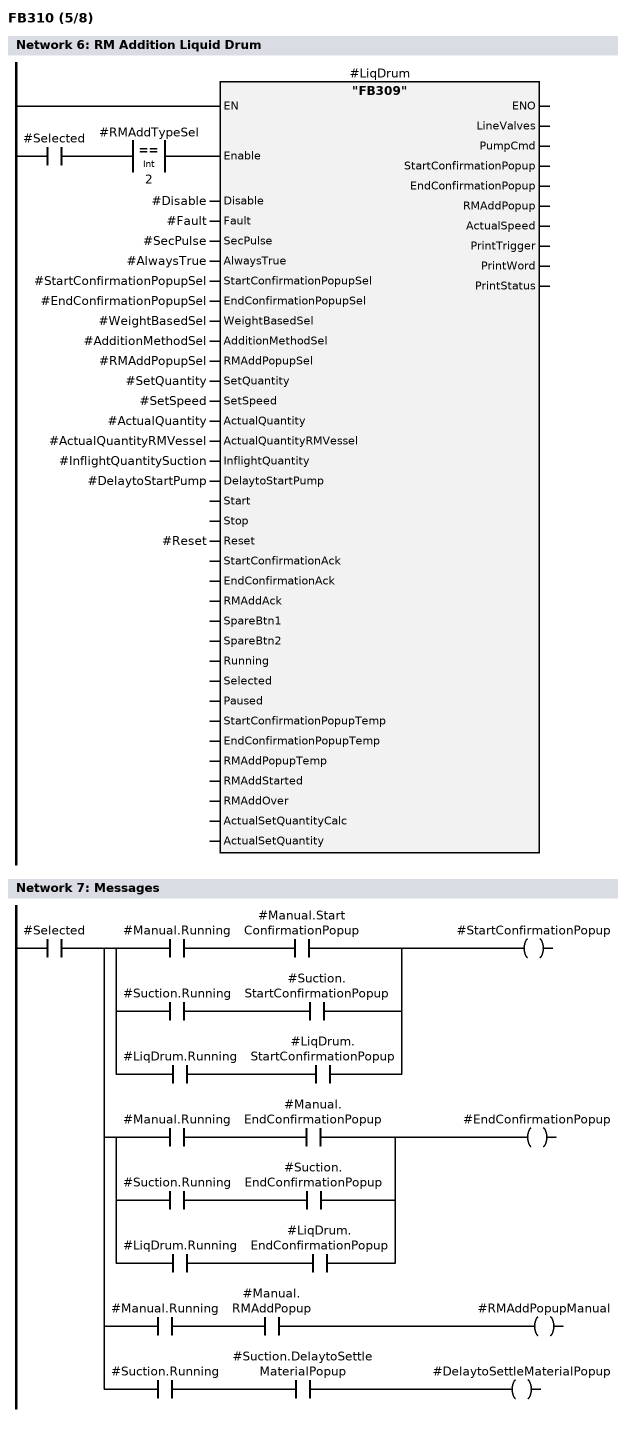
   RUNG wire#powerrail
      #LiqDrum(Enable := wire#w1, Disable := #Disable, Fault := #Fault, SecPulse := #SecPulse, AlwaysTrue := #AlwaysTrue, StartConfirmationPopupSel := #StartConfirmationPopupSel, EndConfirmationPopupSel := #EndConfirmationPopupSel, WeightBasedSel := #WeightBasedSel, AdditionMethodSel := #AdditionMethodSel, RMAddPopupSel := #RMAddPopupSel, SetQuantity := #SetQuantity, SetSpeed := #SetSpeed, ActualQuantity := #ActualQuantity, ActualQuantityRMVessel := #ActualQuantityRMVessel, InflightQuantity := #InflightQuantitySuction, DelaytoStartPump := #DelaytoStartPump, Start :=, Stop :=, Reset := #Reset, StartConfirmationAck :=, EndConfirmationAck :=, RMAddAck :=, SpareBtn1 :=, SpareBtn2 :=, Running :=, Selected :=, Paused :=, StartConfirmationPopupTemp :=, EndConfirmationPopupTemp :=, RMAddPopupTemp :=, RMAddStarted :=, RMAddOver :=, ActualSetQuantityCalc :=, ActualSetQuantity :=, LineValves =>, PumpCmd =>, StartConfirmationPopup =>, EndConfirmationPopup =>, RMAddPopup =>, ActualSpeed =>, PrintTrigger =>, PrintWord =>, PrintStatus =>)
   END_RUNG
   RUNG wire#powerrail
      Contact( #Selected )
      { S7_Templates := "SrcType := Int" } EQ_Contact(in1 := #RMAddTypeSel, in2 := 2)
   END_RUNG wire#w1
   // the same network as SCL:
   #LiqDrum(Enable := #Selected AND (#RMAddTypeSel = 2),   // "FB309"
            Disable := #Disable,
            Fault := #Fault,
            SecPulse := #SecPulse,
            AlwaysTrue := #AlwaysTrue,
            StartConfirmationPopupSel := #StartConfirmationPopupSel,
            EndConfirmationPopupSel := #EndConfirmationPopupSel,
            WeightBasedSel := #WeightBasedSel,
            AdditionMethodSel := #AdditionMethodSel,
            RMAddPopupSel := #RMAddPopupSel,
            SetQuantity := #SetQuantity,
            SetSpeed := #SetSpeed,
            ActualQuantity := #ActualQuantity,
            ActualQuantityRMVessel := #ActualQuantityRMVessel,
            InflightQuantity := #InflightQuantitySuction,
            DelaytoStartPump := #DelaytoStartPump,
            Reset := #Reset);
END_REGION

REGION Network 7: Messages
   RUNG wire#powerrail
      Contact( #Selected )
      wire#w1
      Contact( #Manual.Running )
      Contact( #Manual.StartConfirmationPopup )
      wire#w2
      Coil( #StartConfirmationPopup )
   END_RUNG
   RUNG wire#w1
      Contact( #Suction.Running )
      Contact( #Suction.StartConfirmationPopup )
   END_RUNG wire#w2
   RUNG wire#w1
      Contact( #LiqDrum.Running )
      Contact( #LiqDrum.StartConfirmationPopup )
   END_RUNG wire#w2
   RUNG wire#w1
      Contact( #Manual.Running )
      Contact( #Manual.EndConfirmationPopup )
      wire#w3
      Coil( #EndConfirmationPopup )
   END_RUNG
   RUNG wire#w1
      Contact( #Suction.Running )
      Contact( #Suction.EndConfirmationPopup )
   END_RUNG wire#w3
   RUNG wire#w1
      Contact( #LiqDrum.Running )
      Contact( #LiqDrum.EndConfirmationPopup )
   END_RUNG wire#w3
   RUNG wire#w1
      Contact( #Manual.Running )
      Contact( #Manual.RMAddPopup )
      Coil( #RMAddPopupManual )
   END_RUNG
   RUNG wire#w1
      Contact( #Suction.Running )
      Contact( #Suction.DelaytoSettleMaterialPopup )
      Coil( #DelaytoSettleMaterialPopup )
   END_RUNG
   // the same network as SCL:
   #StartConfirmationPopup := #Selected AND ((#Manual.Running AND #Manual.StartConfirmationPopup) OR (#Suction.Running AND #Suction.StartConfirmationPopup) OR (#LiqDrum.Running AND #LiqDrum.StartConfirmationPopup));
   #EndConfirmationPopup := #Selected AND ((#Manual.Running AND #Manual.EndConfirmationPopup) OR (#Suction.Running AND #Suction.EndConfirmationPopup) OR (#LiqDrum.Running AND #LiqDrum.EndConfirmationPopup));
   #RMAddPopupManual := #Selected AND #Manual.Running AND #Manual.RMAddPopup;
   #DelaytoSettleMaterialPopup := #Selected AND #Suction.Running AND #Suction.DelaytoSettleMaterialPopup;
END_REGION

REGION Network 8: Output
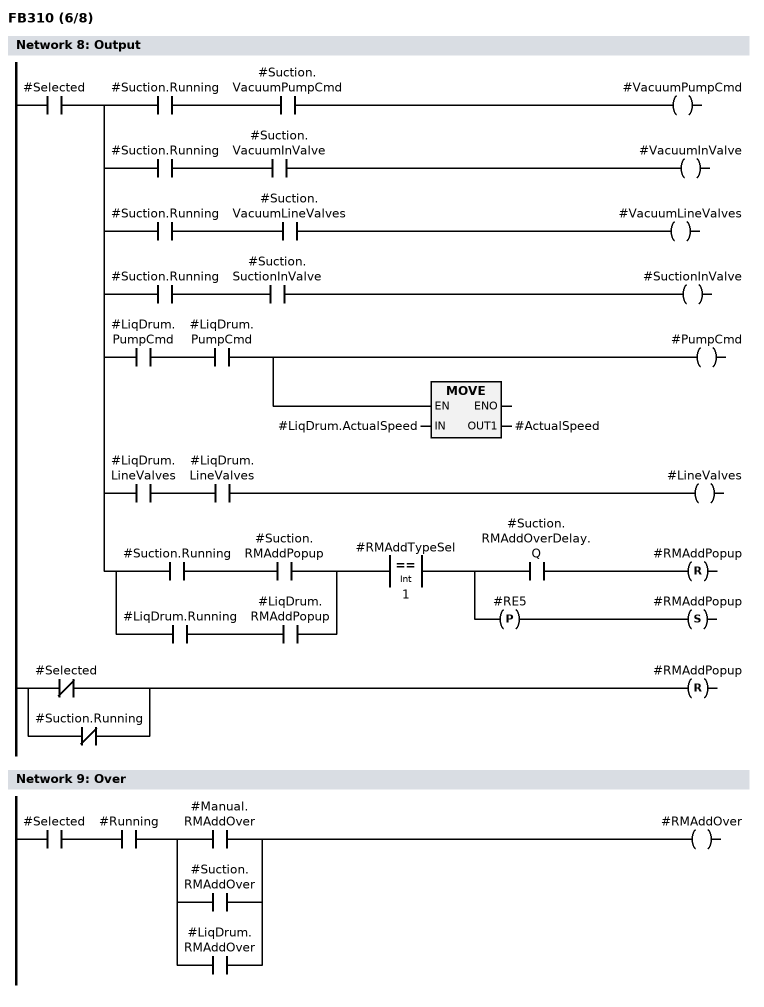
   RUNG wire#powerrail
      Contact( #Selected )
      wire#w1
      Contact( #Suction.Running )
      Contact( #Suction.VacuumPumpCmd )
      Coil( #VacuumPumpCmd )
   END_RUNG
   RUNG wire#w1
      Contact( #Suction.Running )
      Contact( #Suction.VacuumInValve )
      Coil( #VacuumInValve )
   END_RUNG
   RUNG wire#w1
      Contact( #Suction.Running )
      Contact( #Suction.VacuumLineValves )
      Coil( #VacuumLineValves )
   END_RUNG
   RUNG wire#w1
      Contact( #Suction.Running )
      Contact( #Suction.SuctionInValve )
      Coil( #SuctionInValve )
   END_RUNG
   RUNG wire#w1
      Contact( #LiqDrum.PumpCmd )
      Contact( #LiqDrum.PumpCmd )
      wire#w2
      Coil( #PumpCmd )
   END_RUNG
   RUNG wire#w2
      Move(in := #LiqDrum.ActualSpeed, out1 => #ActualSpeed)
   END_RUNG
   RUNG wire#w1
      Contact( #LiqDrum.LineValves )
      Contact( #LiqDrum.LineValves )
      Coil( #LineValves )
   END_RUNG
   RUNG wire#w1
      Contact( #Suction.Running )
      Contact( #Suction.RMAddPopup )
      wire#w3
      { S7_Templates := "SrcType := Int" } EQ_Contact(in1 := #RMAddTypeSel, in2 := 1)
      wire#w4
      Contact( #Suction.RMAddOverDelay.Q )
      R_Coil( #RMAddPopup )
   END_RUNG
   RUNG wire#w1
      Contact( #LiqDrum.Running )
      Contact( #LiqDrum.RMAddPopup )
   END_RUNG wire#w3
   RUNG wire#w4
      P_Trig( #RE5 )
      S_Coil( #RMAddPopup )
   END_RUNG
   RUNG wire#powerrail
      I_Contact( #Selected )
      wire#w5
      R_Coil( #RMAddPopup )
   END_RUNG
   RUNG wire#powerrail
      I_Contact( #Suction.Running )
   END_RUNG wire#w5
   // the same network as SCL:
   #VacuumPumpCmd := #Selected AND #Suction.Running AND #Suction.VacuumPumpCmd;
   #VacuumInValve := #Selected AND #Suction.Running AND #Suction.VacuumInValve;
   #VacuumLineValves := #Selected AND #Suction.Running AND #Suction.VacuumLineValves;
   #SuctionInValve := #Selected AND #Suction.Running AND #Suction.SuctionInValve;
   #PumpCmd := #Selected AND #LiqDrum.PumpCmd AND #LiqDrum.PumpCmd;
   IF #PumpCmd THEN #ActualSpeed := #LiqDrum.ActualSpeed; END_IF;
   #LineValves := #Selected AND #LiqDrum.LineValves AND #LiqDrum.LineValves;
   #_w1 := #Selected AND ((#Suction.Running AND #Suction.RMAddPopup) OR (#LiqDrum.Running AND #LiqDrum.RMAddPopup)) AND (#RMAddTypeSel = 1);
   IF #_w1 AND #Suction.RMAddOverDelay.Q THEN #RMAddPopup := FALSE; END_IF;
   #_w2 := #_w1 AND NOT #RE5;   // rising edge
   #RE5 := #_w1;
   IF #_w2 THEN #RMAddPopup := TRUE; END_IF;
   IF NOT #Selected OR NOT #Suction.Running THEN #RMAddPopup := FALSE; END_IF;
END_REGION

REGION Network 9: Over
   RUNG wire#powerrail
      Contact( #Selected )
      Contact( #Running )
      wire#w1
      Contact( #Manual.RMAddOver )
      wire#w2
      Coil( #RMAddOver )
   END_RUNG
   RUNG wire#w1
      Contact( #Suction.RMAddOver )
   END_RUNG wire#w2
   RUNG wire#w1
      Contact( #LiqDrum.RMAddOver )
   END_RUNG wire#w2
   // the same network as SCL:
   #RMAddOver := #Selected AND #Running AND (#Manual.RMAddOver OR #Suction.RMAddOver OR #LiqDrum.RMAddOver);
END_REGION

REGION Network 10: Print Status
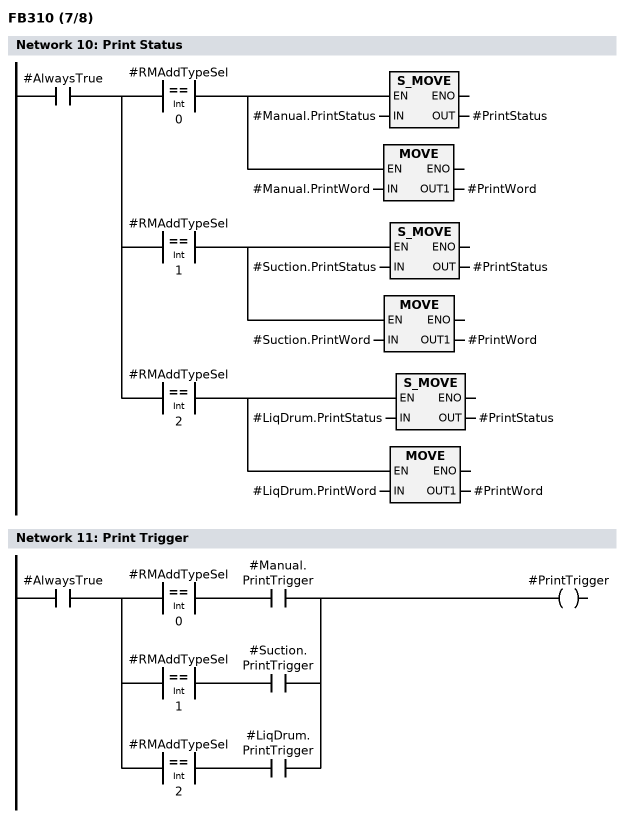
   RUNG wire#powerrail
      Contact( #AlwaysTrue )
      wire#w1
      { S7_Templates := "SrcType := Int" } EQ_Contact(in1 := #RMAddTypeSel, in2 := 0)
      wire#w2
      S_Move(in := #Manual.PrintStatus, out => #PrintStatus)
   END_RUNG
   RUNG wire#w2
      Move(in := #Manual.PrintWord, out1 => #PrintWord)
   END_RUNG
   RUNG wire#w1
      { S7_Templates := "SrcType := Int" } EQ_Contact(in1 := #RMAddTypeSel, in2 := 1)
      wire#w3
      S_Move(in := #Suction.PrintStatus, out => #PrintStatus)
   END_RUNG
   RUNG wire#w3
      Move(in := #Suction.PrintWord, out1 => #PrintWord)
   END_RUNG
   RUNG wire#w1
      { S7_Templates := "SrcType := Int" } EQ_Contact(in1 := #RMAddTypeSel, in2 := 2)
      wire#w4
      S_Move(in := #LiqDrum.PrintStatus, out => #PrintStatus)
   END_RUNG
   RUNG wire#w4
      Move(in := #LiqDrum.PrintWord, out1 => #PrintWord)
   END_RUNG
   // the same network as SCL:
   IF #AlwaysTrue AND (#RMAddTypeSel = 0) THEN
       #PrintStatus := #Manual.PrintStatus;
       #PrintWord := #Manual.PrintWord;
   END_IF;
   IF #AlwaysTrue AND (#RMAddTypeSel = 1) THEN
       #PrintStatus := #Suction.PrintStatus;
       #PrintWord := #Suction.PrintWord;
   END_IF;
   IF #AlwaysTrue AND (#RMAddTypeSel = 2) THEN
       #PrintStatus := #LiqDrum.PrintStatus;
       #PrintWord := #LiqDrum.PrintWord;
   END_IF;
END_REGION

REGION Network 11: Print Trigger
   RUNG wire#powerrail
      Contact( #AlwaysTrue )
      wire#w1
      { S7_Templates := "SrcType := Int" } EQ_Contact(in1 := #RMAddTypeSel, in2 := 0)
      Contact( #Manual.PrintTrigger )
      wire#w2
      Coil( #PrintTrigger )
   END_RUNG
   RUNG wire#w1
      { S7_Templates := "SrcType := Int" } EQ_Contact(in1 := #RMAddTypeSel, in2 := 1)
      Contact( #Suction.PrintTrigger )
   END_RUNG wire#w2
   RUNG wire#w1
      { S7_Templates := "SrcType := Int" } EQ_Contact(in1 := #RMAddTypeSel, in2 := 2)
      Contact( #LiqDrum.PrintTrigger )
   END_RUNG wire#w2
   // the same network as SCL:
   #PrintTrigger := #AlwaysTrue AND (((#RMAddTypeSel = 0) AND #Manual.PrintTrigger) OR ((#RMAddTypeSel = 1) AND #Suction.PrintTrigger) OR ((#RMAddTypeSel = 2) AND #LiqDrum.PrintTrigger));
END_REGION

REGION Network 12: Button Reset
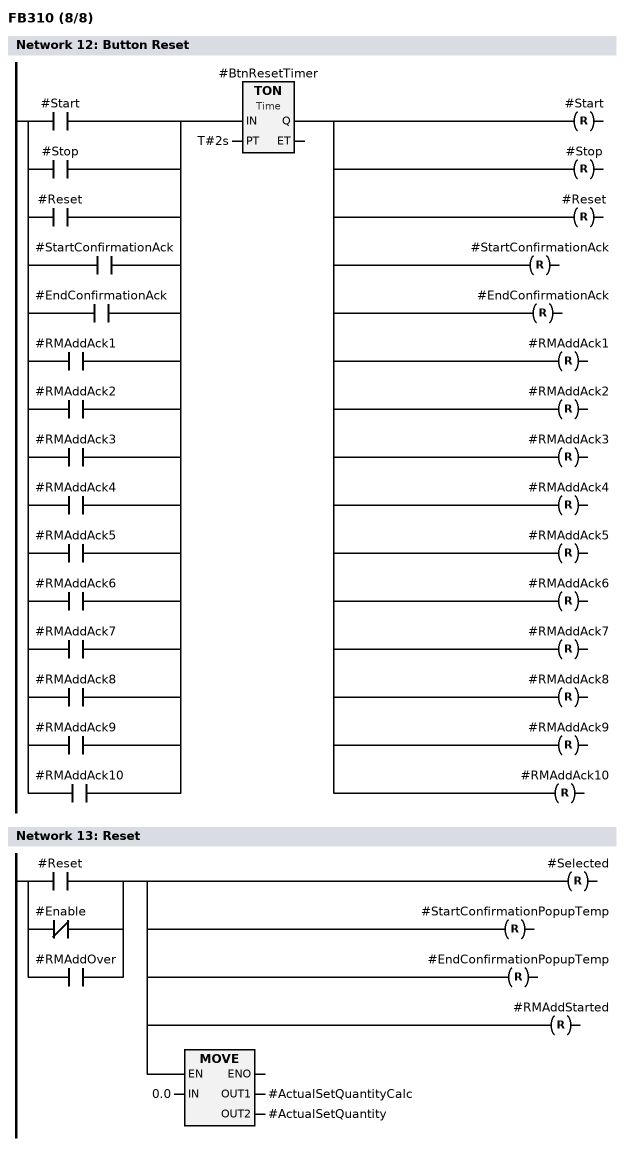
   RUNG wire#powerrail
      Contact( #Start )
      wire#w1
      { S7_Templates := "time_type := Time" } #BtnResetTimer.TON(pt := T#2s, et =>)
      wire#w2
      R_Coil( #Start )
   END_RUNG
   RUNG wire#powerrail
      Contact( #Stop )
   END_RUNG wire#w1
   RUNG wire#powerrail
      Contact( #Reset )
   END_RUNG wire#w1
   RUNG wire#powerrail
      Contact( #StartConfirmationAck )
   END_RUNG wire#w1
   RUNG wire#powerrail
      Contact( #EndConfirmationAck )
   END_RUNG wire#w1
   RUNG wire#powerrail
      Contact( #RMAddAck1 )
   END_RUNG wire#w1
   RUNG wire#powerrail
      Contact( #RMAddAck2 )
   END_RUNG wire#w1
   RUNG wire#powerrail
      Contact( #RMAddAck3 )
   END_RUNG wire#w1
   RUNG wire#powerrail
      Contact( #RMAddAck4 )
   END_RUNG wire#w1
   RUNG wire#powerrail
      Contact( #RMAddAck5 )
   END_RUNG wire#w1
   RUNG wire#powerrail
      Contact( #RMAddAck6 )
   END_RUNG wire#w1
   RUNG wire#powerrail
      Contact( #RMAddAck7 )
   END_RUNG wire#w1
   RUNG wire#powerrail
      Contact( #RMAddAck8 )
   END_RUNG wire#w1
   RUNG wire#powerrail
      Contact( #RMAddAck9 )
   END_RUNG wire#w1
   RUNG wire#powerrail
      Contact( #RMAddAck10 )
   END_RUNG wire#w1
   RUNG wire#w2
      R_Coil( #Stop )
   END_RUNG
   RUNG wire#w2
      R_Coil( #Reset )
   END_RUNG
   RUNG wire#w2
      R_Coil( #StartConfirmationAck )
   END_RUNG
   RUNG wire#w2
      R_Coil( #EndConfirmationAck )
   END_RUNG
   RUNG wire#w2
      R_Coil( #RMAddAck1 )
   END_RUNG
   RUNG wire#w2
      R_Coil( #RMAddAck2 )
   END_RUNG
   RUNG wire#w2
      R_Coil( #RMAddAck3 )
   END_RUNG
   RUNG wire#w2
      R_Coil( #RMAddAck4 )
   END_RUNG
   RUNG wire#w2
      R_Coil( #RMAddAck5 )
   END_RUNG
   RUNG wire#w2
      R_Coil( #RMAddAck6 )
   END_RUNG
   RUNG wire#w2
      R_Coil( #RMAddAck7 )
   END_RUNG
   RUNG wire#w2
      R_Coil( #RMAddAck8 )
   END_RUNG
   RUNG wire#w2
      R_Coil( #RMAddAck9 )
   END_RUNG
   RUNG wire#w2
      R_Coil( #RMAddAck10 )
   END_RUNG
   // the same network as SCL:
   #BtnResetTimer(IN := #Start OR #Stop OR #Reset OR #StartConfirmationAck OR #EndConfirmationAck OR #RMAddAck1 OR #RMAddAck2 OR #RMAddAck3 OR #RMAddAck4 OR #RMAddAck5 OR #RMAddAck6 OR #RMAddAck7 OR #RMAddAck8 OR #RMAddAck9 OR #RMAddAck10,   // TON
                  PT := T#2s);
   IF #BtnResetTimer.Q THEN
       #Start := FALSE;
       #Stop := FALSE;
       #Reset := FALSE;
       #StartConfirmationAck := FALSE;
       #EndConfirmationAck := FALSE;
       #RMAddAck1 := FALSE;
       #RMAddAck2 := FALSE;
       #RMAddAck3 := FALSE;
       #RMAddAck4 := FALSE;
       #RMAddAck5 := FALSE;
       #RMAddAck6 := FALSE;
       #RMAddAck7 := FALSE;
       #RMAddAck8 := FALSE;
       #RMAddAck9 := FALSE;
       #RMAddAck10 := FALSE;
   END_IF;
END_REGION

REGION Network 13: Reset
   RUNG wire#powerrail
      Contact( #Reset )
      wire#w1
      R_Coil( #Selected )
   END_RUNG
   RUNG wire#powerrail
      I_Contact( #Enable )
   END_RUNG wire#w1
   RUNG wire#powerrail
      Contact( #RMAddOver )
   END_RUNG wire#w1
   RUNG wire#w1
      R_Coil( #StartConfirmationPopupTemp )
   END_RUNG
   RUNG wire#w1
      R_Coil( #EndConfirmationPopupTemp )
   END_RUNG
   RUNG wire#w1
      R_Coil( #RMAddStarted )
   END_RUNG
   RUNG wire#w1
      Move(in := 0.0, out1 => #ActualSetQuantityCalc, out2 => #ActualSetQuantity)
   END_RUNG
   // the same network as SCL:
   IF #Reset OR NOT #Enable OR #RMAddOver THEN
       #Selected := FALSE;
       #StartConfirmationPopupTemp := FALSE;
       #EndConfirmationPopupTemp := FALSE;
       #RMAddStarted := FALSE;
       #ActualSetQuantityCalc := 0.0;
       #ActualSetQuantity := 0.0;
   END_IF;
END_REGION
END_FUNCTION_BLOCK

FUNCTION_BLOCK "FB307"   // FB307, LAD
TITLE = FB307
{ S7_Optimized_Access := 'FALSE' }
AUTHOR : PRECISE
FAMILY : PRECISE
// RAW MATERIAL ADDITION MANUAL
// stored: AutoNumber false, SetENOAutomatically false
   VAR_INPUT
      Enable : Bool;
      Disable : Bool;
      Fault : Bool;
      SecPulse : Bool;
      AlwaysTrue : Bool;
      StartConfirmationPopupSel : Bool;   // StartConfirmationPopupSel: 0-NO/1-YES
      EndConfirmationPopupSel : Bool;   // EndConfirmationPopupSel: 0-NO/1-YES
      MixingTimerDone : Bool;
      SetRMNo : Int := 1;   // Max-10
      VesselSafetyPressure : Real;
      VesselActPressure : Real;
   END_VAR
   VAR_OUTPUT
      StartConfirmationPopup : Bool;   // For Start Confirmation Popup Selection: Yes
      EndConfirmationPopup : Bool;   // For End Confirmation Popup Selection: Yes
      RMAddPopup : Bool;
      VisibleRM1 : Bool;
      VisibleRM2 : Bool;
      VisibleRM3 : Bool;
      VisibleRM4 : Bool;
      VisibleRM5 : Bool;
      VisibleRM6 : Bool;
      VisibleRM7 : Bool;
      VisibleRM8 : Bool;
      VisibleRM9 : Bool;
      VisibleRM10 : Bool;
      PrintTrigger : Bool;
      MixerCmd : Bool;
      PrintWord : Int;
      PrintStatus : String[50];
      VesselUnderPressure : Bool;
   END_VAR
   VAR_IN_OUT
      Start : Bool;
      Stop : Bool;
      Reset : Bool;
      StartConfirmationAck : Bool;   // For Start Confirmation Popup Selection: Yes
      EndConfirmationAck : Bool;   // For End Confirmation Popup Selection: Yes
      AckRM1 : Bool;
      AckRM2 : Bool;
      AckRM3 : Bool;
      AckRM4 : Bool;
      AckRM5 : Bool;
      AckRM6 : Bool;
      AckRM7 : Bool;
      AckRM8 : Bool;
      AckRM9 : Bool;
      AckRM10 : Bool;
      Running : Bool;
      Selected : Bool;
      Paused : Bool;
      StartConfirmationPopupTemp : Bool;   // For Start Confirmation Popup Selection: Yes
      EndConfirmationPopupTemp : Bool;   // For End Confirmation Popup Selection: Yes
      RMAddStarted : Bool;
      RMAddOver : Bool;
      AddDoneRM1 : Bool;
      AddDoneRM2 : Bool;
      AddDoneRM3 : Bool;
      AddDoneRM4 : Bool;
      AddDoneRM5 : Bool;
      AddDoneRM6 : Bool;
      AddDoneRM7 : Bool;
      AddDoneRM8 : Bool;
      AddDoneRM9 : Bool;
      AddDoneRM10 : Bool;
   END_VAR
   VAR
      PrintTriggerTemp : Bool;
      RE1 : Bool;
      RE2 : Bool;
      RE3 : Bool;
      RE4 : Bool;
      RE5 : Bool;
      RE6 : Bool;
      RE7 : Bool;
      RE8 : Bool;
      RE9 : Bool;
      RE10 : Bool;
      RE11 : Bool;
      RE12 : Bool;
      RE13 : Bool;
      RE14 : Bool;
      RE15 : Bool;
      RE16 : Bool;
      RE17 : Bool;
      PrintTriggerResetTimer { S7_SetPoint := 'True'} : TON_TIME;
      BtnResetTimer { S7_SetPoint := 'True'} : TON_TIME;
      RMAddOverDelay { S7_SetPoint := 'True'} : TON_TIME;
      NameRM1 : String[100];
      NameRM2 : String[100];
      NameRM3 : String[100];
      NameRM4 : String[100];
      NameRM5 : String[100];
      NameRM6 : String[100];
      NameRM7 : String[100];
      NameRM8 : String[100];
      NameRM9 : String[100];
      NameRM10 : String[100];
   END_VAR
   VAR_TEMP
      STATUS1 : String[40];
      STATUS2 : String[40];
      STATUS3 : String[40];
      STATUS4 : String[40];
      STATUS5 : String[40];
      STATUS6 : String[40];
      STATUS7 : String[40];
      STATUS8 : String[40];
      STATUS9 : String[40];
      STATUS10 : String[40];
      Blank : String[40];
   END_VAR
   VAR_TEMP   // added for the SCL form of the ladder/FBD networks
      _w1 : Bool;
      _w2 : Bool;
      _w3 : Bool;
      _w4 : Bool;
      _w5 : Bool;
      _w6 : Bool;
      _w7 : Bool;
      _w8 : Bool;
      _w9 : Bool;
      _w10 : Bool;
      _w11 : Bool;
      _w12 : Bool;
      _w13 : Bool;
      _w14 : Bool;
      _w15 : Bool;
      _w16 : Bool;
      _w17 : Bool;
      _w18 : Bool;
      _w19 : Bool;
      _w20 : Bool;
      _w21 : Bool;
      _w22 : Bool;
      _w23 : Bool;
      _w24 : Bool;
      _w25 : Bool;
   END_VAR
BEGIN

REGION Network 1: Running
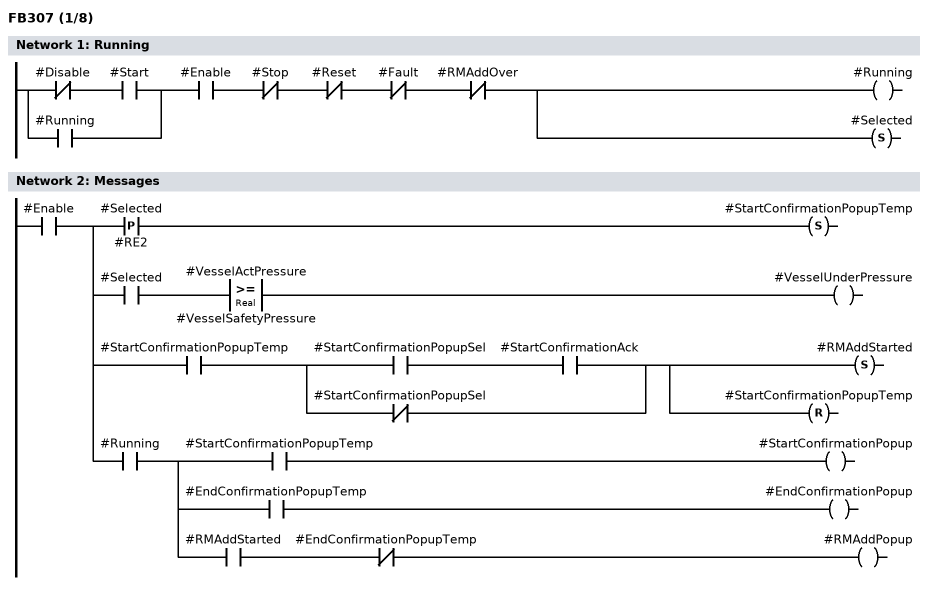
   RUNG wire#powerrail
      I_Contact( #Disable )
      Contact( #Start )
      wire#w1
      Contact( #Enable )
      I_Contact( #Stop )
      I_Contact( #Reset )
      I_Contact( #Fault )
      I_Contact( #RMAddOver )
      wire#w2
      Coil( #Running )
   END_RUNG
   RUNG wire#powerrail
      Contact( #Running )
   END_RUNG wire#w1
   RUNG wire#w2
      S_Coil( #Selected )
   END_RUNG
   // the same network as SCL:
   #Running := ((NOT #Disable AND #Start) OR #Running) AND #Enable AND NOT #Stop AND NOT #Reset AND NOT #Fault AND NOT #RMAddOver;
   IF #Running THEN #Selected := TRUE; END_IF;
END_REGION

REGION Network 2: Messages
   RUNG wire#powerrail
      Contact( #Enable )
      wire#w1
      P_Contact(operand := #Selected, bit := #RE2)
      S_Coil( #StartConfirmationPopupTemp )
   END_RUNG
   RUNG wire#w1
      Contact( #Selected )
      { S7_Templates := "SrcType := Real" } GE_Contact(in1 := #VesselActPressure, in2 := #VesselSafetyPressure)
      Coil( #VesselUnderPressure )
   END_RUNG
   RUNG wire#w1
      Contact( #StartConfirmationPopupTemp )
      wire#w2
      Contact( #StartConfirmationPopupSel )
      Contact( #StartConfirmationAck )
      wire#w3
      S_Coil( #RMAddStarted )
   END_RUNG
   RUNG wire#w2
      I_Contact( #StartConfirmationPopupSel )
   END_RUNG wire#w3
   RUNG wire#w3
      R_Coil( #StartConfirmationPopupTemp )
   END_RUNG
   RUNG wire#w1
      Contact( #Running )
      wire#w4
      Contact( #StartConfirmationPopupTemp )
      Coil( #StartConfirmationPopup )
   END_RUNG
   RUNG wire#w4
      Contact( #EndConfirmationPopupTemp )
      Coil( #EndConfirmationPopup )
   END_RUNG
   RUNG wire#w4
      Contact( #RMAddStarted )
      I_Contact( #EndConfirmationPopupTemp )
      Coil( #RMAddPopup )
   END_RUNG
   // the same network as SCL:
   #_w1 := #Enable AND #Selected AND NOT #RE2;   // rising edge of #Selected
   #RE2 := #Selected;
   IF #_w1 THEN #StartConfirmationPopupTemp := TRUE; END_IF;
   #VesselUnderPressure := #Enable AND #Selected AND (#VesselActPressure >= #VesselSafetyPressure);
   IF #Enable AND #StartConfirmationPopupTemp AND ((#StartConfirmationPopupSel AND #StartConfirmationAck) OR NOT #StartConfirmationPopupSel) THEN
       #RMAddStarted := TRUE;
       #StartConfirmationPopupTemp := FALSE;
   END_IF;
   #_w2 := #Enable AND #Running;
   #StartConfirmationPopup := #_w2 AND #StartConfirmationPopupTemp;
   #EndConfirmationPopup := #_w2 AND #EndConfirmationPopupTemp;
   #RMAddPopup := #_w2 AND #RMAddStarted AND NOT #EndConfirmationPopupTemp;
END_REGION

REGION Network 3: Visibility for RM
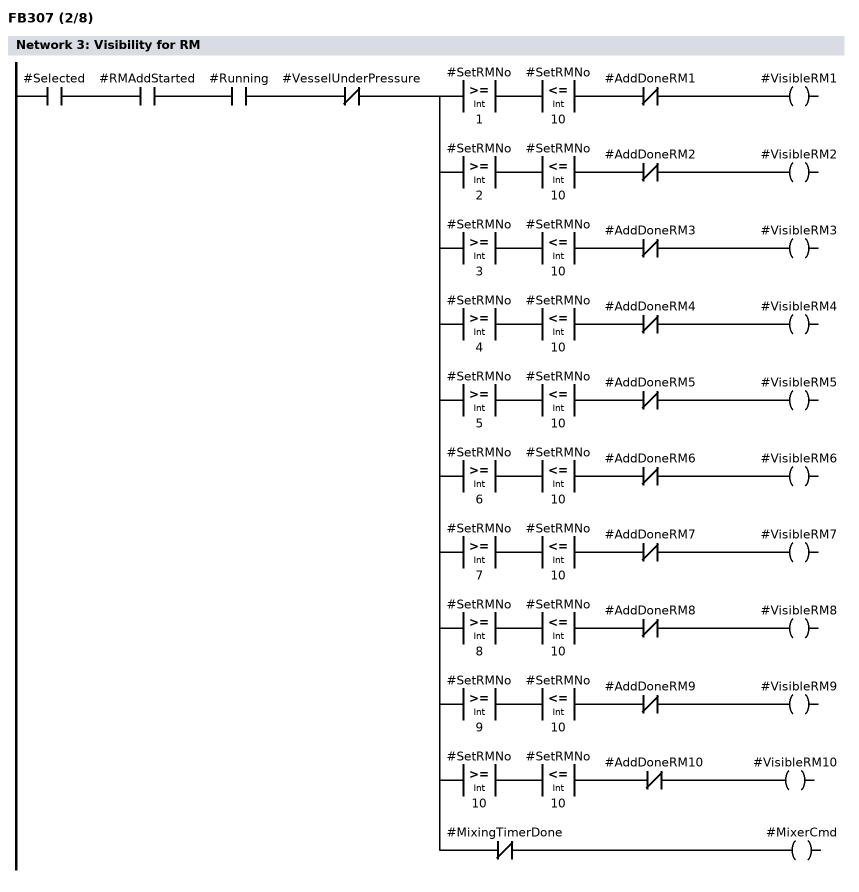
   RUNG wire#powerrail
      Contact( #Selected )
      Contact( #RMAddStarted )
      Contact( #Running )
      I_Contact( #VesselUnderPressure )
      wire#w1
      { S7_Templates := "SrcType := Int" } GE_Contact(in1 := #SetRMNo, in2 := 1)
      { S7_Templates := "SrcType := Int" } LE_Contact(in1 := #SetRMNo, in2 := 10)
      I_Contact( #AddDoneRM1 )
      Coil( #VisibleRM1 )
   END_RUNG
   RUNG wire#w1
      { S7_Templates := "SrcType := Int" } GE_Contact(in1 := #SetRMNo, in2 := 2)
      { S7_Templates := "SrcType := Int" } LE_Contact(in1 := #SetRMNo, in2 := 10)
      I_Contact( #AddDoneRM2 )
      Coil( #VisibleRM2 )
   END_RUNG
   RUNG wire#w1
      { S7_Templates := "SrcType := Int" } GE_Contact(in1 := #SetRMNo, in2 := 3)
      { S7_Templates := "SrcType := Int" } LE_Contact(in1 := #SetRMNo, in2 := 10)
      I_Contact( #AddDoneRM3 )
      Coil( #VisibleRM3 )
   END_RUNG
   RUNG wire#w1
      { S7_Templates := "SrcType := Int" } GE_Contact(in1 := #SetRMNo, in2 := 4)
      { S7_Templates := "SrcType := Int" } LE_Contact(in1 := #SetRMNo, in2 := 10)
      I_Contact( #AddDoneRM4 )
      Coil( #VisibleRM4 )
   END_RUNG
   RUNG wire#w1
      { S7_Templates := "SrcType := Int" } GE_Contact(in1 := #SetRMNo, in2 := 5)
      { S7_Templates := "SrcType := Int" } LE_Contact(in1 := #SetRMNo, in2 := 10)
      I_Contact( #AddDoneRM5 )
      Coil( #VisibleRM5 )
   END_RUNG
   RUNG wire#w1
      { S7_Templates := "SrcType := Int" } GE_Contact(in1 := #SetRMNo, in2 := 6)
      { S7_Templates := "SrcType := Int" } LE_Contact(in1 := #SetRMNo, in2 := 10)
      I_Contact( #AddDoneRM6 )
      Coil( #VisibleRM6 )
   END_RUNG
   RUNG wire#w1
      { S7_Templates := "SrcType := Int" } GE_Contact(in1 := #SetRMNo, in2 := 7)
      { S7_Templates := "SrcType := Int" } LE_Contact(in1 := #SetRMNo, in2 := 10)
      I_Contact( #AddDoneRM7 )
      Coil( #VisibleRM7 )
   END_RUNG
   RUNG wire#w1
      { S7_Templates := "SrcType := Int" } GE_Contact(in1 := #SetRMNo, in2 := 8)
      { S7_Templates := "SrcType := Int" } LE_Contact(in1 := #SetRMNo, in2 := 10)
      I_Contact( #AddDoneRM8 )
      Coil( #VisibleRM8 )
   END_RUNG
   RUNG wire#w1
      { S7_Templates := "SrcType := Int" } GE_Contact(in1 := #SetRMNo, in2 := 9)
      { S7_Templates := "SrcType := Int" } LE_Contact(in1 := #SetRMNo, in2 := 10)
      I_Contact( #AddDoneRM9 )
      Coil( #VisibleRM9 )
   END_RUNG
   RUNG wire#w1
      { S7_Templates := "SrcType := Int" } GE_Contact(in1 := #SetRMNo, in2 := 10)
      { S7_Templates := "SrcType := Int" } LE_Contact(in1 := #SetRMNo, in2 := 10)
      I_Contact( #AddDoneRM10 )
      Coil( #VisibleRM10 )
   END_RUNG
   RUNG wire#w1
      I_Contact( #MixingTimerDone )
      Coil( #MixerCmd )
   END_RUNG
   // the same network as SCL:
   #_w1 := #Selected AND #RMAddStarted AND #Running AND NOT #VesselUnderPressure;
   #VisibleRM1 := #_w1 AND (#SetRMNo >= 1) AND (#SetRMNo <= 10) AND NOT #AddDoneRM1;
   #VisibleRM2 := #_w1 AND (#SetRMNo >= 2) AND (#SetRMNo <= 10) AND NOT #AddDoneRM2;
   #VisibleRM3 := #_w1 AND (#SetRMNo >= 3) AND (#SetRMNo <= 10) AND NOT #AddDoneRM3;
   #VisibleRM4 := #_w1 AND (#SetRMNo >= 4) AND (#SetRMNo <= 10) AND NOT #AddDoneRM4;
   #VisibleRM5 := #_w1 AND (#SetRMNo >= 5) AND (#SetRMNo <= 10) AND NOT #AddDoneRM5;
   #VisibleRM6 := #_w1 AND (#SetRMNo >= 6) AND (#SetRMNo <= 10) AND NOT #AddDoneRM6;
   #VisibleRM7 := #_w1 AND (#SetRMNo >= 7) AND (#SetRMNo <= 10) AND NOT #AddDoneRM7;
   #VisibleRM8 := #_w1 AND (#SetRMNo >= 8) AND (#SetRMNo <= 10) AND NOT #AddDoneRM8;
   #VisibleRM9 := #_w1 AND (#SetRMNo >= 9) AND (#SetRMNo <= 10) AND NOT #AddDoneRM9;
   #VisibleRM10 := #_w1 AND (#SetRMNo >= 10) AND (#SetRMNo <= 10) AND NOT #AddDoneRM10;
   #MixerCmd := #_w1 AND NOT #MixingTimerDone;
END_REGION

REGION Network 4: Add Done
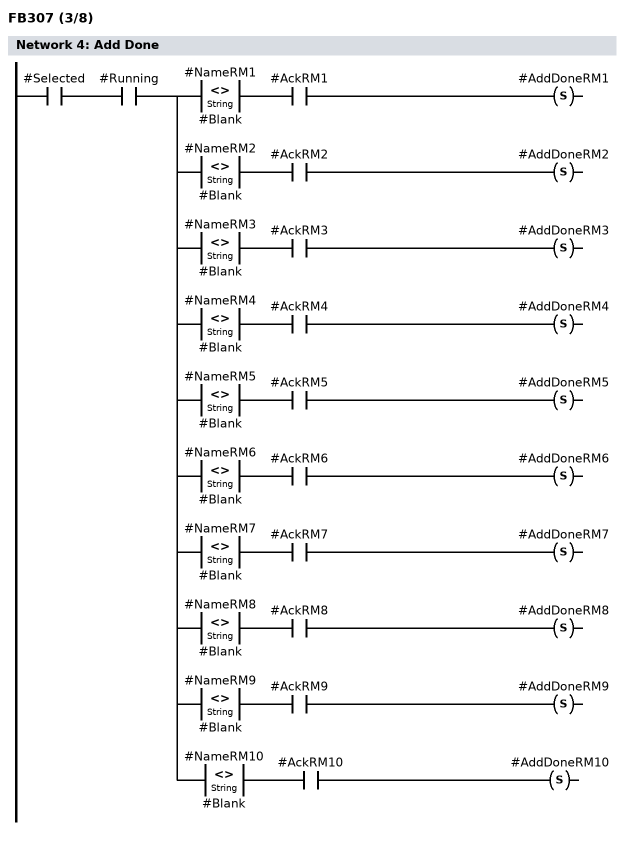
   RUNG wire#powerrail
      Contact( #Selected )
      Contact( #Running )
      wire#w1
      { S7_Templates := "SrcType := String" } NE_Contact(in1 := #NameRM1, in2 := #Blank)
      Contact( #AckRM1 )
      S_Coil( #AddDoneRM1 )
   END_RUNG
   RUNG wire#w1
      { S7_Templates := "SrcType := String" } NE_Contact(in1 := #NameRM2, in2 := #Blank)
      Contact( #AckRM2 )
      S_Coil( #AddDoneRM2 )
   END_RUNG
   RUNG wire#w1
      { S7_Templates := "SrcType := String" } NE_Contact(in1 := #NameRM3, in2 := #Blank)
      Contact( #AckRM3 )
      S_Coil( #AddDoneRM3 )
   END_RUNG
   RUNG wire#w1
      { S7_Templates := "SrcType := String" } NE_Contact(in1 := #NameRM4, in2 := #Blank)
      Contact( #AckRM4 )
      S_Coil( #AddDoneRM4 )
   END_RUNG
   RUNG wire#w1
      { S7_Templates := "SrcType := String" } NE_Contact(in1 := #NameRM5, in2 := #Blank)
      Contact( #AckRM5 )
      S_Coil( #AddDoneRM5 )
   END_RUNG
   RUNG wire#w1
      { S7_Templates := "SrcType := String" } NE_Contact(in1 := #NameRM6, in2 := #Blank)
      Contact( #AckRM6 )
      S_Coil( #AddDoneRM6 )
   END_RUNG
   RUNG wire#w1
      { S7_Templates := "SrcType := String" } NE_Contact(in1 := #NameRM7, in2 := #Blank)
      Contact( #AckRM7 )
      S_Coil( #AddDoneRM7 )
   END_RUNG
   RUNG wire#w1
      { S7_Templates := "SrcType := String" } NE_Contact(in1 := #NameRM8, in2 := #Blank)
      Contact( #AckRM8 )
      S_Coil( #AddDoneRM8 )
   END_RUNG
   RUNG wire#w1
      { S7_Templates := "SrcType := String" } NE_Contact(in1 := #NameRM9, in2 := #Blank)
      Contact( #AckRM9 )
      S_Coil( #AddDoneRM9 )
   END_RUNG
   RUNG wire#w1
      { S7_Templates := "SrcType := String" } NE_Contact(in1 := #NameRM10, in2 := #Blank)
      Contact( #AckRM10 )
      S_Coil( #AddDoneRM10 )
   END_RUNG
   // the same network as SCL:
   #_w1 := #Selected AND #Running;
   IF #_w1 AND (#NameRM1 <> #Blank) AND #AckRM1 THEN #AddDoneRM1 := TRUE; END_IF;
   IF #_w1 AND (#NameRM2 <> #Blank) AND #AckRM2 THEN #AddDoneRM2 := TRUE; END_IF;
   IF #_w1 AND (#NameRM3 <> #Blank) AND #AckRM3 THEN #AddDoneRM3 := TRUE; END_IF;
   IF #_w1 AND (#NameRM4 <> #Blank) AND #AckRM4 THEN #AddDoneRM4 := TRUE; END_IF;
   IF #_w1 AND (#NameRM5 <> #Blank) AND #AckRM5 THEN #AddDoneRM5 := TRUE; END_IF;
   IF #_w1 AND (#NameRM6 <> #Blank) AND #AckRM6 THEN #AddDoneRM6 := TRUE; END_IF;
   IF #_w1 AND (#NameRM7 <> #Blank) AND #AckRM7 THEN #AddDoneRM7 := TRUE; END_IF;
   IF #_w1 AND (#NameRM8 <> #Blank) AND #AckRM8 THEN #AddDoneRM8 := TRUE; END_IF;
   IF #_w1 AND (#NameRM9 <> #Blank) AND #AckRM9 THEN #AddDoneRM9 := TRUE; END_IF;
   IF #_w1 AND (#NameRM10 <> #Blank) AND #AckRM10 THEN #AddDoneRM10 := TRUE; END_IF;
END_REGION

REGION Network 5: All Addition Done
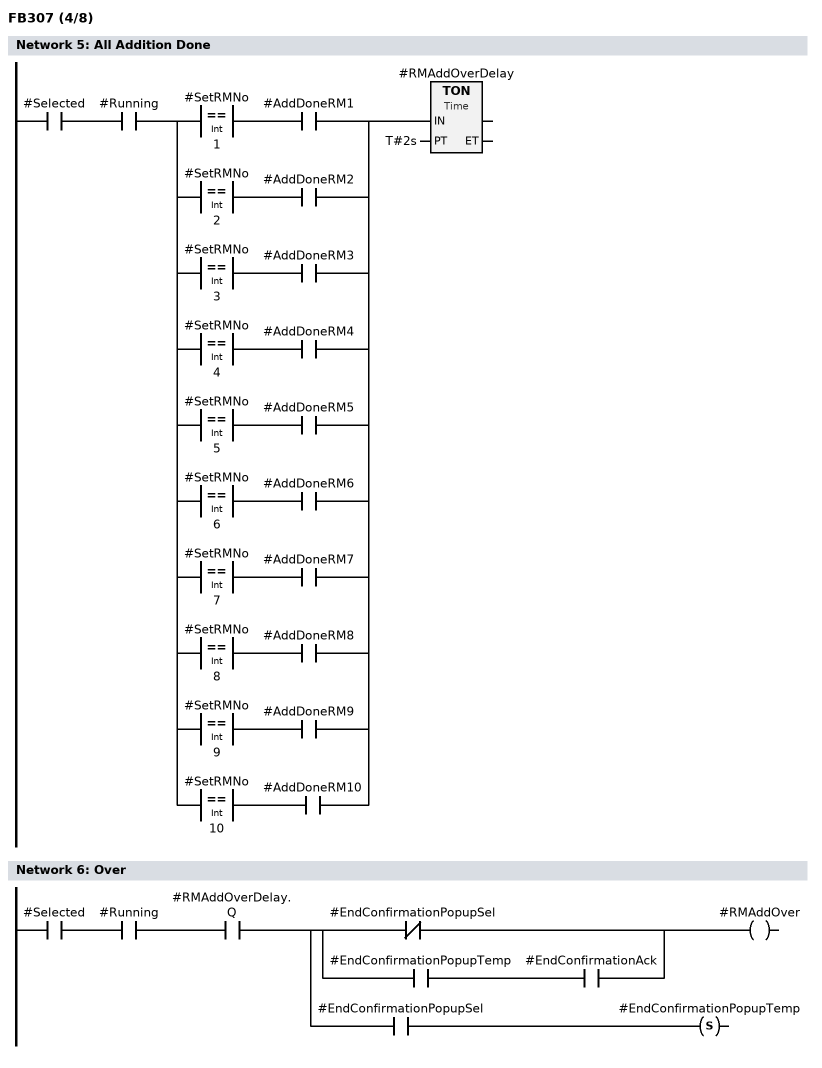
   RUNG wire#powerrail
      Contact( #Selected )
      Contact( #Running )
      wire#w1
      { S7_Templates := "SrcType := Int" } EQ_Contact(in1 := #SetRMNo, in2 := 1)
      Contact( #AddDoneRM1 )
      wire#w2
      { S7_Templates := "time_type := Time" } #RMAddOverDelay.TON(pt := T#2s, et =>)
   END_RUNG
   RUNG wire#w1
      { S7_Templates := "SrcType := Int" } EQ_Contact(in1 := #SetRMNo, in2 := 2)
      Contact( #AddDoneRM2 )
   END_RUNG wire#w2
   RUNG wire#w1
      { S7_Templates := "SrcType := Int" } EQ_Contact(in1 := #SetRMNo, in2 := 3)
      Contact( #AddDoneRM3 )
   END_RUNG wire#w2
   RUNG wire#w1
      { S7_Templates := "SrcType := Int" } EQ_Contact(in1 := #SetRMNo, in2 := 4)
      Contact( #AddDoneRM4 )
   END_RUNG wire#w2
   RUNG wire#w1
      { S7_Templates := "SrcType := Int" } EQ_Contact(in1 := #SetRMNo, in2 := 5)
      Contact( #AddDoneRM5 )
   END_RUNG wire#w2
   RUNG wire#w1
      { S7_Templates := "SrcType := Int" } EQ_Contact(in1 := #SetRMNo, in2 := 6)
      Contact( #AddDoneRM6 )
   END_RUNG wire#w2
   RUNG wire#w1
      { S7_Templates := "SrcType := Int" } EQ_Contact(in1 := #SetRMNo, in2 := 7)
      Contact( #AddDoneRM7 )
   END_RUNG wire#w2
   RUNG wire#w1
      { S7_Templates := "SrcType := Int" } EQ_Contact(in1 := #SetRMNo, in2 := 8)
      Contact( #AddDoneRM8 )
   END_RUNG wire#w2
   RUNG wire#w1
      { S7_Templates := "SrcType := Int" } EQ_Contact(in1 := #SetRMNo, in2 := 9)
      Contact( #AddDoneRM9 )
   END_RUNG wire#w2
   RUNG wire#w1
      { S7_Templates := "SrcType := Int" } EQ_Contact(in1 := #SetRMNo, in2 := 10)
      Contact( #AddDoneRM10 )
   END_RUNG wire#w2
   // the same network as SCL:
   #RMAddOverDelay(IN := #Selected AND #Running AND (((#SetRMNo = 1) AND #AddDoneRM1) OR ((#SetRMNo = 2) AND #AddDoneRM2) OR ((#SetRMNo = 3) AND #AddDoneRM3) OR ((#SetRMNo = 4) AND #AddDoneRM4) OR ((#SetRMNo = 5) AND #AddDoneRM5) OR ((#SetRMNo = 6) AND #AddDoneRM6) OR ((#SetRMNo = 7) AND #AddDoneRM7) OR ((#SetRMNo = 8) AND #AddDoneRM8) OR ((#SetRMNo = 9) AND #AddDoneRM9) OR ((#SetRMNo = 10) AND #AddDoneRM10)),   // TON
                   PT := T#2s);
END_REGION

REGION Network 6: Over
   RUNG wire#powerrail
      Contact( #Selected )
      Contact( #Running )
      Contact( #RMAddOverDelay.Q )
      wire#w1
      I_Contact( #EndConfirmationPopupSel )
      wire#w2
      Coil( #RMAddOver )
   END_RUNG
   RUNG wire#w1
      Contact( #EndConfirmationPopupTemp )
      Contact( #EndConfirmationAck )
   END_RUNG wire#w2
   RUNG wire#w1
      Contact( #EndConfirmationPopupSel )
      S_Coil( #EndConfirmationPopupTemp )
   END_RUNG
   // the same network as SCL:
   #_w1 := #Selected AND #Running AND #RMAddOverDelay.Q;
   #RMAddOver := #_w1 AND (NOT #EndConfirmationPopupSel OR (#EndConfirmationPopupTemp AND #EndConfirmationAck));
   IF #_w1 AND #EndConfirmationPopupSel THEN #EndConfirmationPopupTemp := TRUE; END_IF;
END_REGION

REGION Network 7: Event Status
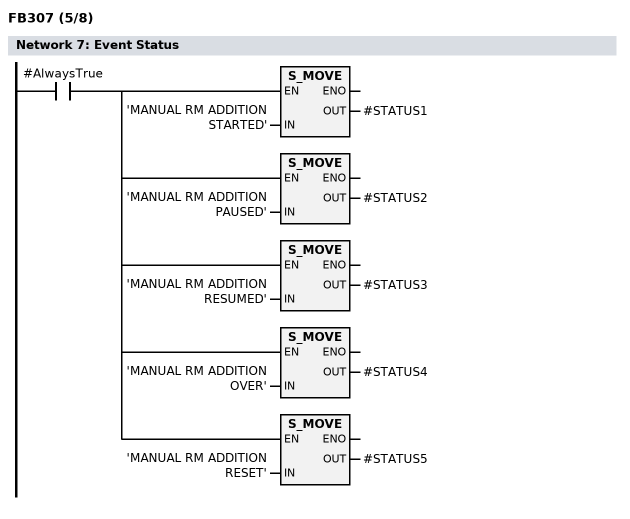
   RUNG wire#powerrail
      Contact( #AlwaysTrue )
      wire#w1
      S_Move(in := 'MANUAL RM ADDITION STARTED', out => #STATUS1)
   END_RUNG
   RUNG wire#w1
      S_Move(in := 'MANUAL RM ADDITION PAUSED', out => #STATUS2)
   END_RUNG
   RUNG wire#w1
      S_Move(in := 'MANUAL RM ADDITION RESUMED', out => #STATUS3)
   END_RUNG
   RUNG wire#w1
      S_Move(in := 'MANUAL RM ADDITION OVER', out => #STATUS4)
   END_RUNG
   RUNG wire#w1
      S_Move(in := 'MANUAL RM ADDITION RESET', out => #STATUS5)
   END_RUNG
   // the same network as SCL:
   IF #AlwaysTrue THEN
       #STATUS1 := 'MANUAL RM ADDITION STARTED';
       #STATUS2 := 'MANUAL RM ADDITION PAUSED';
       #STATUS3 := 'MANUAL RM ADDITION RESUMED';
       #STATUS4 := 'MANUAL RM ADDITION OVER';
       #STATUS5 := 'MANUAL RM ADDITION RESET';
   END_IF;
END_REGION

REGION Network 8: Print Logic
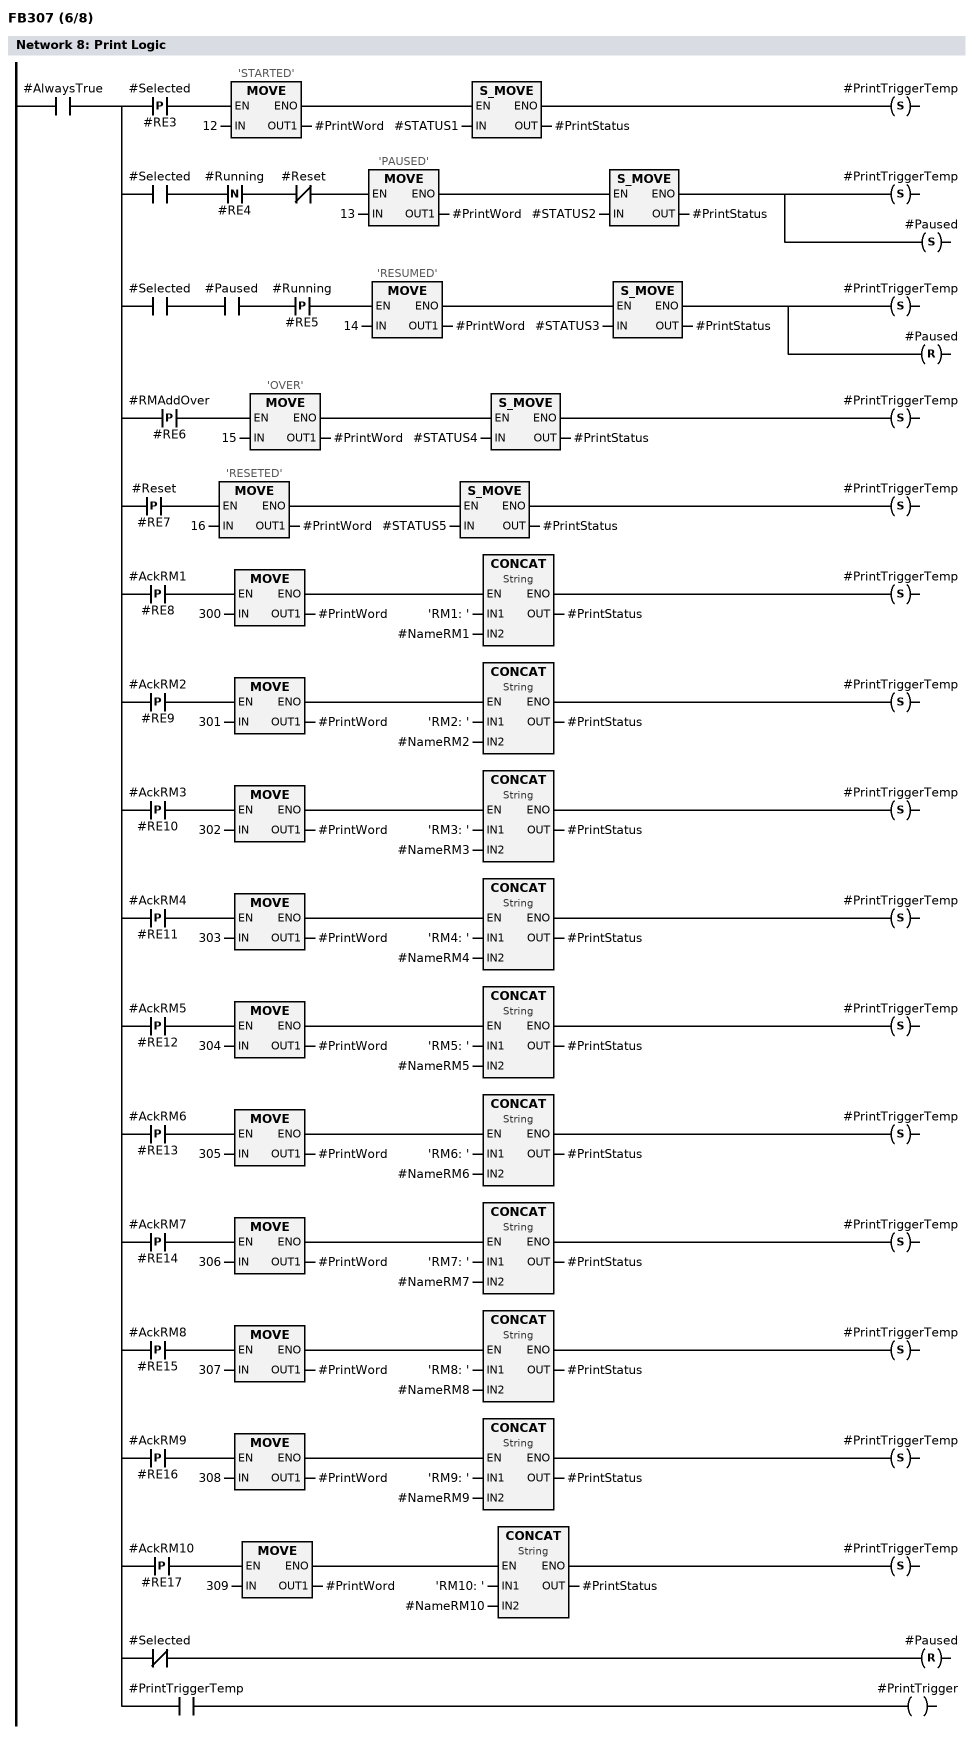
   RUNG wire#powerrail
      Contact( #AlwaysTrue )
      wire#w1
      P_Contact(operand := #Selected, bit := #RE3)
      { S7_GenerateENO := "TRUE" } Move(in := 12, out1 => #PrintWord)   // 'STARTED'
      S_Move(in := #STATUS1, out => #PrintStatus)
      S_Coil( #PrintTriggerTemp )
   END_RUNG
   RUNG wire#w1
      Contact( #Selected )
      N_Contact(operand := #Running, bit := #RE4)
      I_Contact( #Reset )
      { S7_GenerateENO := "TRUE" } Move(in := 13, out1 => #PrintWord)   // 'PAUSED'
      S_Move(in := #STATUS2, out => #PrintStatus)
      wire#w2
      S_Coil( #PrintTriggerTemp )
   END_RUNG
   RUNG wire#w2
      S_Coil( #Paused )
   END_RUNG
   RUNG wire#w1
      Contact( #Selected )
      Contact( #Paused )
      P_Contact(operand := #Running, bit := #RE5)
      { S7_GenerateENO := "TRUE" } Move(in := 14, out1 => #PrintWord)   // 'RESUMED'
      S_Move(in := #STATUS3, out => #PrintStatus)
      wire#w3
      S_Coil( #PrintTriggerTemp )
   END_RUNG
   RUNG wire#w3
      R_Coil( #Paused )
   END_RUNG
   RUNG wire#w1
      P_Contact(operand := #RMAddOver, bit := #RE6)
      { S7_GenerateENO := "TRUE" } Move(in := 15, out1 => #PrintWord)   // 'OVER'
      S_Move(in := #STATUS4, out => #PrintStatus)
      S_Coil( #PrintTriggerTemp )
   END_RUNG
   RUNG wire#w1
      P_Contact(operand := #Reset, bit := #RE7)
      { S7_GenerateENO := "TRUE" } Move(in := 16, out1 => #PrintWord)   // 'RESETED'
      S_Move(in := #STATUS5, out => #PrintStatus)
      S_Coil( #PrintTriggerTemp )
   END_RUNG
   RUNG wire#w1
      P_Contact(operand := #AckRM1, bit := #RE8)
      { S7_GenerateENO := "TRUE" } Move(in := 300, out1 => #PrintWord)
      { S7_Templates := "[card := 2, str_type := String]" } CONCAT(IN1 := 'RM1: ', IN2 := #NameRM1, OUT => #PrintStatus)
      S_Coil( #PrintTriggerTemp )
   END_RUNG
   RUNG wire#w1
      P_Contact(operand := #AckRM2, bit := #RE9)
      { S7_GenerateENO := "TRUE" } Move(in := 301, out1 => #PrintWord)
      { S7_Templates := "[card := 2, str_type := String]" } CONCAT(IN1 := 'RM2: ', IN2 := #NameRM2, OUT => #PrintStatus)
      S_Coil( #PrintTriggerTemp )
   END_RUNG
   RUNG wire#w1
      P_Contact(operand := #AckRM3, bit := #RE10)
      { S7_GenerateENO := "TRUE" } Move(in := 302, out1 => #PrintWord)
      { S7_Templates := "[card := 2, str_type := String]" } CONCAT(IN1 := 'RM3: ', IN2 := #NameRM3, OUT => #PrintStatus)
      S_Coil( #PrintTriggerTemp )
   END_RUNG
   RUNG wire#w1
      P_Contact(operand := #AckRM4, bit := #RE11)
      { S7_GenerateENO := "TRUE" } Move(in := 303, out1 => #PrintWord)
      { S7_Templates := "[card := 2, str_type := String]" } CONCAT(IN1 := 'RM4: ', IN2 := #NameRM4, OUT => #PrintStatus)
      S_Coil( #PrintTriggerTemp )
   END_RUNG
   RUNG wire#w1
      P_Contact(operand := #AckRM5, bit := #RE12)
      { S7_GenerateENO := "TRUE" } Move(in := 304, out1 => #PrintWord)
      { S7_Templates := "[card := 2, str_type := String]" } CONCAT(IN1 := 'RM5: ', IN2 := #NameRM5, OUT => #PrintStatus)
      S_Coil( #PrintTriggerTemp )
   END_RUNG
   RUNG wire#w1
      P_Contact(operand := #AckRM6, bit := #RE13)
      { S7_GenerateENO := "TRUE" } Move(in := 305, out1 => #PrintWord)
      { S7_Templates := "[card := 2, str_type := String]" } CONCAT(IN1 := 'RM6: ', IN2 := #NameRM6, OUT => #PrintStatus)
      S_Coil( #PrintTriggerTemp )
   END_RUNG
   RUNG wire#w1
      P_Contact(operand := #AckRM7, bit := #RE14)
      { S7_GenerateENO := "TRUE" } Move(in := 306, out1 => #PrintWord)
      { S7_Templates := "[card := 2, str_type := String]" } CONCAT(IN1 := 'RM7: ', IN2 := #NameRM7, OUT => #PrintStatus)
      S_Coil( #PrintTriggerTemp )
   END_RUNG
   RUNG wire#w1
      P_Contact(operand := #AckRM8, bit := #RE15)
      { S7_GenerateENO := "TRUE" } Move(in := 307, out1 => #PrintWord)
      { S7_Templates := "[card := 2, str_type := String]" } CONCAT(IN1 := 'RM8: ', IN2 := #NameRM8, OUT => #PrintStatus)
      S_Coil( #PrintTriggerTemp )
   END_RUNG
   RUNG wire#w1
      P_Contact(operand := #AckRM9, bit := #RE16)
      { S7_GenerateENO := "TRUE" } Move(in := 308, out1 => #PrintWord)
      { S7_Templates := "[card := 2, str_type := String]" } CONCAT(IN1 := 'RM9: ', IN2 := #NameRM9, OUT => #PrintStatus)
      S_Coil( #PrintTriggerTemp )
   END_RUNG
   RUNG wire#w1
      P_Contact(operand := #AckRM10, bit := #RE17)
      { S7_GenerateENO := "TRUE" } Move(in := 309, out1 => #PrintWord)
      { S7_Templates := "[card := 2, str_type := String]" } CONCAT(IN1 := 'RM10: ', IN2 := #NameRM10, OUT => #PrintStatus)
      S_Coil( #PrintTriggerTemp )
   END_RUNG
   RUNG wire#w1
      I_Contact( #Selected )
      R_Coil( #Paused )
   END_RUNG
   RUNG wire#w1
      Contact( #PrintTriggerTemp )
      Coil( #PrintTrigger )
   END_RUNG
   // the same network as SCL:
   // ENO of a box is taken as its EN; it also drops when the box reports an error
   #_w1 := #AlwaysTrue AND #Selected AND NOT #RE3;   // rising edge of #Selected
   #RE3 := #Selected;
   IF #_w1 THEN
       #PrintWord := 12;   // 'STARTED'
       #PrintStatus := #STATUS1;
       #PrintTriggerTemp := TRUE;
   END_IF;
   #_w2 := #AlwaysTrue AND #Selected AND NOT #Running AND #RE4;   // falling edge of #Running
   #RE4 := #Running;
   IF #_w2 AND NOT #Reset THEN
       #PrintWord := 13;   // 'PAUSED'
       #PrintStatus := #STATUS2;
       #PrintTriggerTemp := TRUE;
       #Paused := TRUE;
   END_IF;
   #_w3 := #AlwaysTrue AND #Selected AND #Paused AND #Running AND NOT #RE5;   // rising edge of #Running
   #RE5 := #Running;
   IF #_w3 THEN
       #PrintWord := 14;   // 'RESUMED'
       #PrintStatus := #STATUS3;
       #PrintTriggerTemp := TRUE;
       #Paused := FALSE;
   END_IF;
   #_w4 := #AlwaysTrue AND #RMAddOver AND NOT #RE6;   // rising edge of #RMAddOver
   #RE6 := #RMAddOver;
   IF #_w4 THEN
       #PrintWord := 15;   // 'OVER'
       #PrintStatus := #STATUS4;
       #PrintTriggerTemp := TRUE;
   END_IF;
   #_w5 := #AlwaysTrue AND #Reset AND NOT #RE7;   // rising edge of #Reset
   #RE7 := #Reset;
   IF #_w5 THEN
       #PrintWord := 16;   // 'RESETED'
       #PrintStatus := #STATUS5;
       #PrintTriggerTemp := TRUE;
   END_IF;
   #_w6 := #AlwaysTrue AND #AckRM1 AND NOT #RE8;   // rising edge of #AckRM1
   #RE8 := #AckRM1;
   IF #_w6 THEN #PrintWord := 300; END_IF;
   CONCAT(EN := #_w6, IN1 := 'RM1: ', IN2 := #NameRM1, OUT => #PrintStatus, ENO => #_w7);
   IF #_w7 THEN #PrintTriggerTemp := TRUE; END_IF;
   #_w8 := #AlwaysTrue AND #AckRM2 AND NOT #RE9;   // rising edge of #AckRM2
   #RE9 := #AckRM2;
   IF #_w8 THEN #PrintWord := 301; END_IF;
   CONCAT(EN := #_w8, IN1 := 'RM2: ', IN2 := #NameRM2, OUT => #PrintStatus, ENO => #_w9);
   IF #_w9 THEN #PrintTriggerTemp := TRUE; END_IF;
   #_w10 := #AlwaysTrue AND #AckRM3 AND NOT #RE10;   // rising edge of #AckRM3
   #RE10 := #AckRM3;
   IF #_w10 THEN #PrintWord := 302; END_IF;
   CONCAT(EN := #_w10, IN1 := 'RM3: ', IN2 := #NameRM3, OUT => #PrintStatus, ENO => #_w11);
   IF #_w11 THEN #PrintTriggerTemp := TRUE; END_IF;
   #_w12 := #AlwaysTrue AND #AckRM4 AND NOT #RE11;   // rising edge of #AckRM4
   #RE11 := #AckRM4;
   IF #_w12 THEN #PrintWord := 303; END_IF;
   CONCAT(EN := #_w12, IN1 := 'RM4: ', IN2 := #NameRM4, OUT => #PrintStatus, ENO => #_w13);
   IF #_w13 THEN #PrintTriggerTemp := TRUE; END_IF;
   #_w14 := #AlwaysTrue AND #AckRM5 AND NOT #RE12;   // rising edge of #AckRM5
   #RE12 := #AckRM5;
   IF #_w14 THEN #PrintWord := 304; END_IF;
   CONCAT(EN := #_w14, IN1 := 'RM5: ', IN2 := #NameRM5, OUT => #PrintStatus, ENO => #_w15);
   IF #_w15 THEN #PrintTriggerTemp := TRUE; END_IF;
   #_w16 := #AlwaysTrue AND #AckRM6 AND NOT #RE13;   // rising edge of #AckRM6
   #RE13 := #AckRM6;
   IF #_w16 THEN #PrintWord := 305; END_IF;
   CONCAT(EN := #_w16, IN1 := 'RM6: ', IN2 := #NameRM6, OUT => #PrintStatus, ENO => #_w17);
   IF #_w17 THEN #PrintTriggerTemp := TRUE; END_IF;
   #_w18 := #AlwaysTrue AND #AckRM7 AND NOT #RE14;   // rising edge of #AckRM7
   #RE14 := #AckRM7;
   IF #_w18 THEN #PrintWord := 306; END_IF;
   CONCAT(EN := #_w18, IN1 := 'RM7: ', IN2 := #NameRM7, OUT => #PrintStatus, ENO => #_w19);
   IF #_w19 THEN #PrintTriggerTemp := TRUE; END_IF;
   #_w20 := #AlwaysTrue AND #AckRM8 AND NOT #RE15;   // rising edge of #AckRM8
   #RE15 := #AckRM8;
   IF #_w20 THEN #PrintWord := 307; END_IF;
   CONCAT(EN := #_w20, IN1 := 'RM8: ', IN2 := #NameRM8, OUT => #PrintStatus, ENO => #_w21);
   IF #_w21 THEN #PrintTriggerTemp := TRUE; END_IF;
   #_w22 := #AlwaysTrue AND #AckRM9 AND NOT #RE16;   // rising edge of #AckRM9
   #RE16 := #AckRM9;
   IF #_w22 THEN #PrintWord := 308; END_IF;
   CONCAT(EN := #_w22, IN1 := 'RM9: ', IN2 := #NameRM9, OUT => #PrintStatus, ENO => #_w23);
   IF #_w23 THEN #PrintTriggerTemp := TRUE; END_IF;
   #_w24 := #AlwaysTrue AND #AckRM10 AND NOT #RE17;   // rising edge of #AckRM10
   #RE17 := #AckRM10;
   IF #_w24 THEN #PrintWord := 309; END_IF;
   CONCAT(EN := #_w24, IN1 := 'RM10: ', IN2 := #NameRM10, OUT => #PrintStatus, ENO => #_w25);
   IF #_w25 THEN #PrintTriggerTemp := TRUE; END_IF;
   IF #AlwaysTrue AND NOT #Selected THEN #Paused := FALSE; END_IF;
   #PrintTrigger := #AlwaysTrue AND #PrintTriggerTemp;
END_REGION

REGION Network 9: Print Trigger Reset
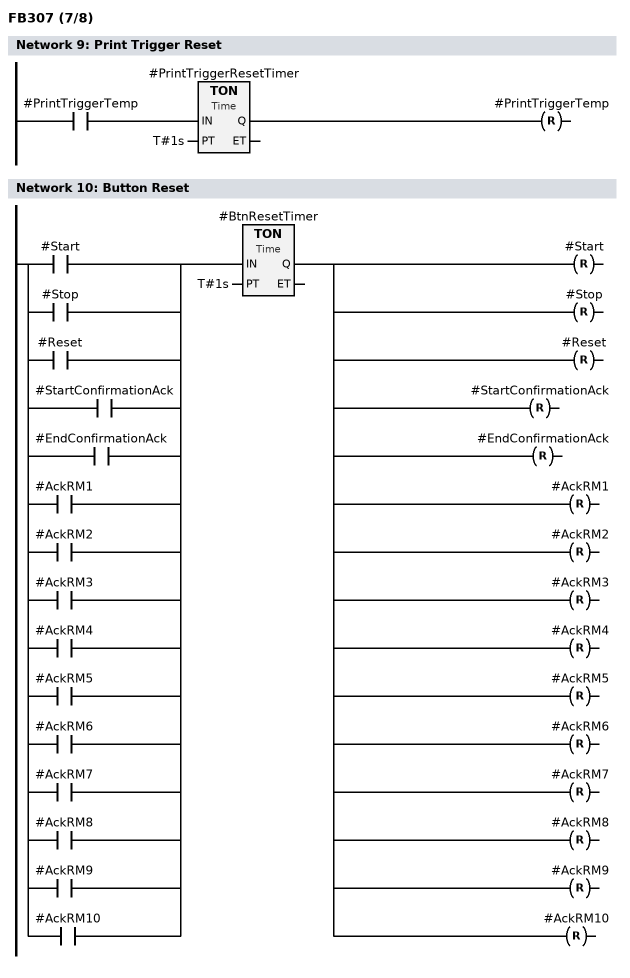
   RUNG wire#powerrail
      Contact( #PrintTriggerTemp )
      { S7_Templates := "time_type := Time" } #PrintTriggerResetTimer.TON(pt := T#1s, et =>)
      R_Coil( #PrintTriggerTemp )
   END_RUNG
   // the same network as SCL:
   #PrintTriggerResetTimer(IN := #PrintTriggerTemp, PT := T#1s);   // TON
   IF #PrintTriggerResetTimer.Q THEN #PrintTriggerTemp := FALSE; END_IF;
END_REGION

REGION Network 10: Button Reset
   RUNG wire#powerrail
      Contact( #Start )
      wire#w1
      { S7_Templates := "time_type := Time" } #BtnResetTimer.TON(pt := T#1s, et =>)
      wire#w2
      R_Coil( #Start )
   END_RUNG
   RUNG wire#powerrail
      Contact( #Stop )
   END_RUNG wire#w1
   RUNG wire#powerrail
      Contact( #Reset )
   END_RUNG wire#w1
   RUNG wire#powerrail
      Contact( #StartConfirmationAck )
   END_RUNG wire#w1
   RUNG wire#powerrail
      Contact( #EndConfirmationAck )
   END_RUNG wire#w1
   RUNG wire#powerrail
      Contact( #AckRM1 )
   END_RUNG wire#w1
   RUNG wire#powerrail
      Contact( #AckRM2 )
   END_RUNG wire#w1
   RUNG wire#powerrail
      Contact( #AckRM3 )
   END_RUNG wire#w1
   RUNG wire#powerrail
      Contact( #AckRM4 )
   END_RUNG wire#w1
   RUNG wire#powerrail
      Contact( #AckRM5 )
   END_RUNG wire#w1
   RUNG wire#powerrail
      Contact( #AckRM6 )
   END_RUNG wire#w1
   RUNG wire#powerrail
      Contact( #AckRM7 )
   END_RUNG wire#w1
   RUNG wire#powerrail
      Contact( #AckRM8 )
   END_RUNG wire#w1
   RUNG wire#powerrail
      Contact( #AckRM9 )
   END_RUNG wire#w1
   RUNG wire#powerrail
      Contact( #AckRM10 )
   END_RUNG wire#w1
   RUNG wire#w2
      R_Coil( #Stop )
   END_RUNG
   RUNG wire#w2
      R_Coil( #Reset )
   END_RUNG
   RUNG wire#w2
      R_Coil( #StartConfirmationAck )
   END_RUNG
   RUNG wire#w2
      R_Coil( #EndConfirmationAck )
   END_RUNG
   RUNG wire#w2
      R_Coil( #AckRM1 )
   END_RUNG
   RUNG wire#w2
      R_Coil( #AckRM2 )
   END_RUNG
   RUNG wire#w2
      R_Coil( #AckRM3 )
   END_RUNG
   RUNG wire#w2
      R_Coil( #AckRM4 )
   END_RUNG
   RUNG wire#w2
      R_Coil( #AckRM5 )
   END_RUNG
   RUNG wire#w2
      R_Coil( #AckRM6 )
   END_RUNG
   RUNG wire#w2
      R_Coil( #AckRM7 )
   END_RUNG
   RUNG wire#w2
      R_Coil( #AckRM8 )
   END_RUNG
   RUNG wire#w2
      R_Coil( #AckRM9 )
   END_RUNG
   RUNG wire#w2
      R_Coil( #AckRM10 )
   END_RUNG
   // the same network as SCL:
   #BtnResetTimer(IN := #Start OR #Stop OR #Reset OR #StartConfirmationAck OR #EndConfirmationAck OR #AckRM1 OR #AckRM2 OR #AckRM3 OR #AckRM4 OR #AckRM5 OR #AckRM6 OR #AckRM7 OR #AckRM8 OR #AckRM9 OR #AckRM10,   // TON
                  PT := T#1s);
   IF #BtnResetTimer.Q THEN
       #Start := FALSE;
       #Stop := FALSE;
       #Reset := FALSE;
       #StartConfirmationAck := FALSE;
       #EndConfirmationAck := FALSE;
       #AckRM1 := FALSE;
       #AckRM2 := FALSE;
       #AckRM3 := FALSE;
       #AckRM4 := FALSE;
       #AckRM5 := FALSE;
       #AckRM6 := FALSE;
       #AckRM7 := FALSE;
       #AckRM8 := FALSE;
       #AckRM9 := FALSE;
       #AckRM10 := FALSE;
   END_IF;
END_REGION

REGION Network 11: Reset
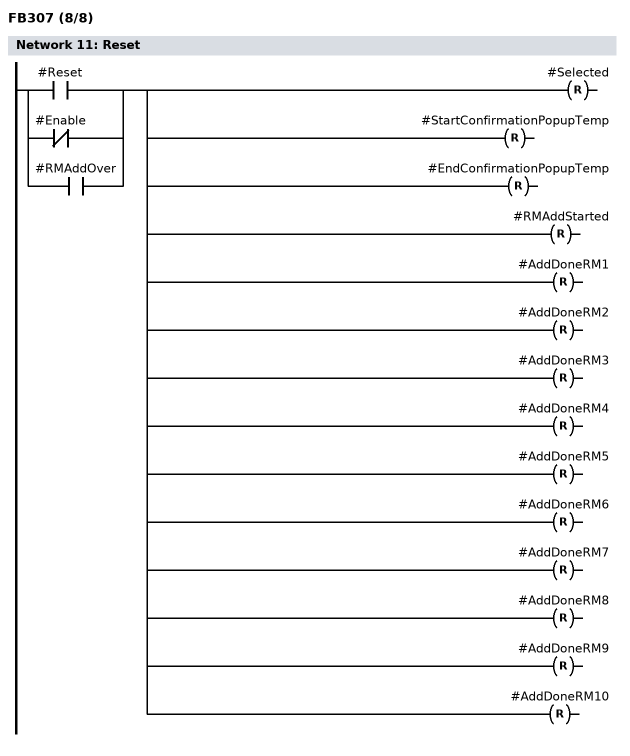
   RUNG wire#powerrail
      Contact( #Reset )
      wire#w1
      R_Coil( #Selected )
   END_RUNG
   RUNG wire#powerrail
      I_Contact( #Enable )
   END_RUNG wire#w1
   RUNG wire#powerrail
      Contact( #RMAddOver )
   END_RUNG wire#w1
   RUNG wire#w1
      R_Coil( #StartConfirmationPopupTemp )
   END_RUNG
   RUNG wire#w1
      R_Coil( #EndConfirmationPopupTemp )
   END_RUNG
   RUNG wire#w1
      R_Coil( #RMAddStarted )
   END_RUNG
   RUNG wire#w1
      R_Coil( #AddDoneRM1 )
   END_RUNG
   RUNG wire#w1
      R_Coil( #AddDoneRM2 )
   END_RUNG
   RUNG wire#w1
      R_Coil( #AddDoneRM3 )
   END_RUNG
   RUNG wire#w1
      R_Coil( #AddDoneRM4 )
   END_RUNG
   RUNG wire#w1
      R_Coil( #AddDoneRM5 )
   END_RUNG
   RUNG wire#w1
      R_Coil( #AddDoneRM6 )
   END_RUNG
   RUNG wire#w1
      R_Coil( #AddDoneRM7 )
   END_RUNG
   RUNG wire#w1
      R_Coil( #AddDoneRM8 )
   END_RUNG
   RUNG wire#w1
      R_Coil( #AddDoneRM9 )
   END_RUNG
   RUNG wire#w1
      R_Coil( #AddDoneRM10 )
   END_RUNG
   // the same network as SCL:
   IF #Reset OR NOT #Enable OR #RMAddOver THEN
       #Selected := FALSE;
       #StartConfirmationPopupTemp := FALSE;
       #EndConfirmationPopupTemp := FALSE;
       #RMAddStarted := FALSE;
       #AddDoneRM1 := FALSE;
       #AddDoneRM2 := FALSE;
       #AddDoneRM3 := FALSE;
       #AddDoneRM4 := FALSE;
       #AddDoneRM5 := FALSE;
       #AddDoneRM6 := FALSE;
       #AddDoneRM7 := FALSE;
       #AddDoneRM8 := FALSE;
       #AddDoneRM9 := FALSE;
       #AddDoneRM10 := FALSE;
   END_IF;
END_REGION
END_FUNCTION_BLOCK

FUNCTION_BLOCK "FB308"   // FB308, LAD
TITLE = FB308
{ S7_Optimized_Access := 'FALSE' }
AUTHOR : PRECISE
FAMILY : PRECISE
// RAW MATERIAL ADDITION SUCTION
// stored: AutoNumber false, SetENOAutomatically false
   VAR_INPUT
      Enable : Bool;
      Disable : Bool;
      Fault : Bool;
      SecPulse : Bool;
      AlwaysTrue : Bool;
      StartConfirmationPopupSel : Bool;   // StartConfirmationPopupSel: 0-NO/1-YES
      EndConfirmationPopupSel : Bool;   // EndConfirmationPopupSel: 0-NO/1-YES
      WeightBasedSel : Bool;   // Weight Based Sel: 0-NO/1-YES
      MixingTimerDone : Bool;
      RMTypeSel : Int;   // RM Type Sel: Graules or Flakes -0/FinePowder-1
      AdditionMethodSel : Bool;   // AdditionMethod : 0-Add In Weight/1-Loss In Weight
      RMAddPopupSel : Bool;   // RM Add Popup Sel: 0-NO/1-YES
      "SetVacuum/SetPressure" : Real := -300.0;   // SetVauum - For unit "mmHg" / SetPressure - For unit "bar"
      SetQuantity : Real := 10.0;   // Weight Based Sel: 1-YES
      "ActualVacuum/ActualPressure" : Real;   // ActualVauum - For unit "mmHg" / ActualPressure - For unit "bar"
      ActualQuantity : Real;   // Collecting Vessel Weight
      ActualQuantityRMVessel : Real;   // Transffering Vessel Weight
      "VacuumTol/PressureTol" : Real := 10.0;   // VacuumTol - For unit "mmHg" / PressureTol - For unit "bar"
      DelaytoSettleMaterial : Int := 5;
      InflightQuantity : Real;
      SetRmNo : Int;
   END_VAR
   VAR_OUTPUT
      VacuumInValve : Bool;
      VacuumLineValves : Bool;
      SuctionInValve : Bool;
      VacuumPumpCmd : Bool;
      StartConfirmationPopup : Bool;   // For Start Confirmation Popup Selection: Yes
      EndConfirmationPopup : Bool;   // For End Confirmation Popup Selection: Yes
      DelaytoSettleMaterialPopup : Bool;   // "WAITING FOR MATERIAL TO SETTLE"
      RMAddPopup : Bool;   // For RMAddPopupSel: 1-YES
      VisibleRM1 : Bool;
      VisibleRM2 : Bool;
      VisibleRM3 : Bool;
      VisibleRM4 : Bool;
      VisibleRM5 : Bool;
      VisibleRM6 : Bool;
      VisibleRM7 : Bool;
      VisibleRM8 : Bool;
      VisibleRM9 : Bool;
      VisibleRM10 : Bool;
      PrintTrigger : Bool;
      MixerCmd : Bool;
      PrintWord : Int;
      PrintStatus : String[50];
   END_VAR
   VAR_IN_OUT
      Start : Bool;
      Stop : Bool;
      Reset : Bool;
      StartConfirmationAck : Bool;   // For Start Confirmation Popup Selection: Yes
      EndConfirmationAck : Bool;   // For End Confirmation Popup Selection: Yes
      RMAddAck1 : Bool;   // For RMAddPopupSel: 1-YES
      SpareBtn1 : Bool;
      SpareBtn2 : Bool;
      Running : Bool;
      Selected : Bool;
      Paused : Bool;
      StartConfirmationPopupTemp : Bool;   // For Start Confirmation Popup Selection: Yes
      EndConfirmationPopupTemp : Bool;   // For End Confirmation Popup Selection: Yes
      DelaytoSettleMaterialPopupTemp : Bool;   // "WAITING FOR MATERIAL TO SETTLE"
      RMAddPopupTemp : Bool;   // For RMAddPopupSel: 1-YES
      RMAddStarted : Bool;
      RMAddOver : Bool;
      VacuumReached : Bool;
      InRange : Bool;
      ActualSetQuantityCalc : Real;   // For WeightBaseSel: 1-YES
      ActualSetQuantity : Real;   // For WeightBaseSel: 1-YES
      "VacuumTolNeg/PressureTolNeg" : Real;   // VacuumTolNeg - For unit "mmHg" / PressureTolNeg - For unit "bar"
      DelaytoSettleMaterialPV : Int;
      RMAddAck2 : Bool;   // For RMAddPopupSel: 1-YES
      RMAddAck3 : Bool;   // For RMAddPopupSel: 1-YES
      RMAddAck4 : Bool;   // For RMAddPopupSel: 1-YES
      RMAddAck5 : Bool;   // For RMAddPopupSel: 1-YES
      RMAddAck6 : Bool;   // For RMAddPopupSel: 1-YES
      RMAddAck7 : Bool;   // For RMAddPopupSel: 1-YES
      RMAddAck8 : Bool;   // For RMAddPopupSel: 1-YES
      RMAddAck9 : Bool;   // For RMAddPopupSel: 1-YES
      RMAddAck10 : Bool;   // For RMAddPopupSel: 1-YES
      AddDoneRM1 : Bool;
      AddDoneRM2 : Bool;
      AddDoneRM3 : Bool;
      AddDoneRM4 : Bool;
      AddDoneRM5 : Bool;
      AddDoneRM6 : Bool;
      AddDoneRM7 : Bool;
      AddDoneRM8 : Bool;
      AddDoneRM9 : Bool;
      AddDoneRM10 : Bool;
      AddDoneRM : Bool;
   END_VAR
   VAR
      PrintTriggerTemp : Bool;
      RE1 : Bool;
      RE2 : Bool;
      RE3 : Bool;
      RE4 : Bool;
      RE5 : Bool;
      RE6 : Bool;
      RE7 : Bool;
      RE8 : Bool;
      PrintTriggerResetTimer { S7_SetPoint := 'True'} : TON_TIME;
      BtnResetTimer { S7_SetPoint := 'True'} : TON_TIME;
      NameRM1 : String[100];
      NameRM2 : String[100];
      NameRM3 : String[100];
      NameRM4 : String[100];
      NameRM5 : String[100];
      NameRM6 : String[100];
      NameRM7 : String[100];
      NameRM8 : String[100];
      NameRM9 : String[100];
      NameRM10 : String[100];
      RMAddOverDelay { S7_SetPoint := 'True'} : TON_TIME;
   END_VAR
   VAR_TEMP
      STATUS1 : String[40];
      STATUS2 : String[40];
      STATUS3 : String[40];
      STATUS4 : String[40];
      STATUS5 : String[40];
      Blank : String[40];
   END_VAR
   VAR_TEMP   // added for the SCL form of the ladder/FBD networks
      _w1 : Bool;
      _w2 : Bool;
      _w3 : Bool;
      _w4 : Bool;
      _w5 : Bool;
      _w6 : Bool;
      _w7 : Bool;
   END_VAR
BEGIN

REGION Network 1: Running
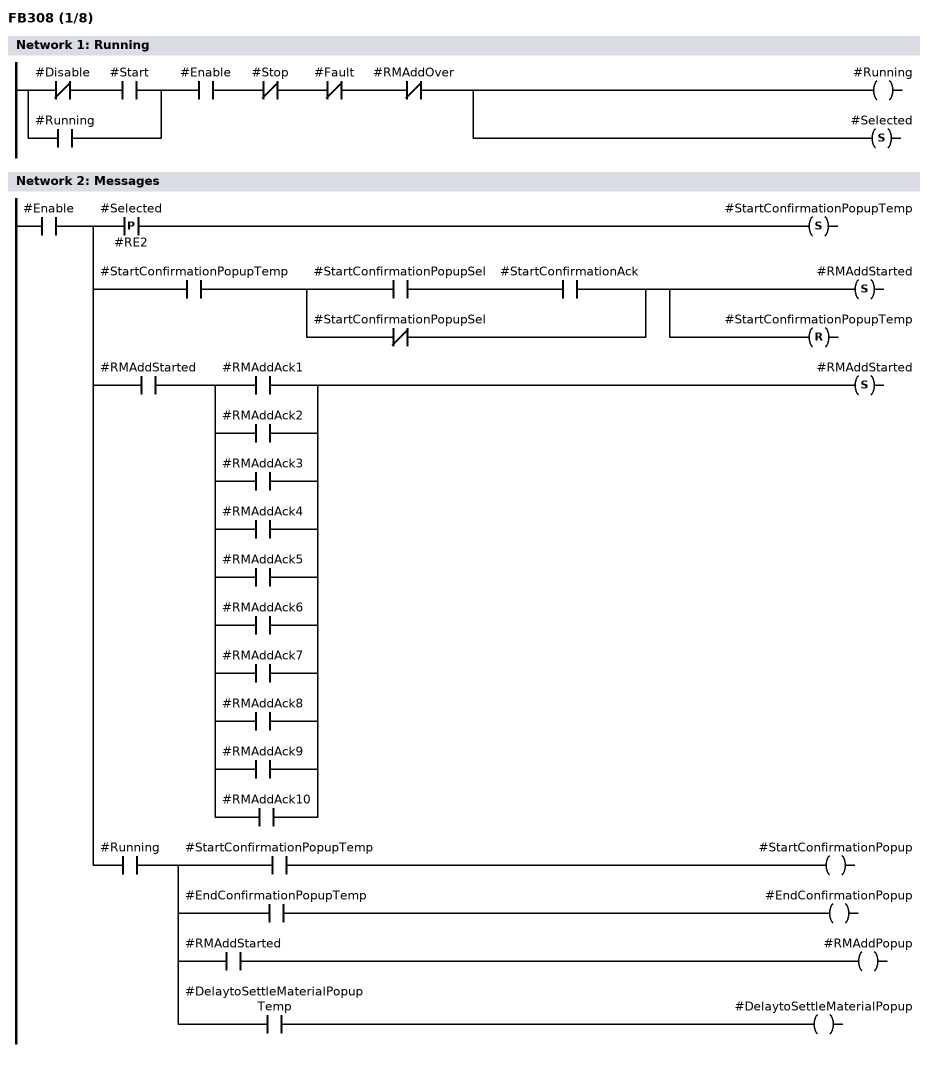
   RUNG wire#powerrail
      I_Contact( #Disable )
      Contact( #Start )
      wire#w1
      Contact( #Enable )
      I_Contact( #Stop )
      I_Contact( #Fault )
      I_Contact( #RMAddOver )
      wire#w2
      Coil( #Running )
   END_RUNG
   RUNG wire#powerrail
      Contact( #Running )
   END_RUNG wire#w1
   RUNG wire#w2
      S_Coil( #Selected )
   END_RUNG
   // the same network as SCL:
   #Running := ((NOT #Disable AND #Start) OR #Running) AND #Enable AND NOT #Stop AND NOT #Fault AND NOT #RMAddOver;
   IF #Running THEN #Selected := TRUE; END_IF;
END_REGION

REGION Network 2: Messages
   RUNG wire#powerrail
      Contact( #Enable )
      wire#w1
      P_Contact(operand := #Selected, bit := #RE2)
      S_Coil( #StartConfirmationPopupTemp )
   END_RUNG
   RUNG wire#w1
      Contact( #StartConfirmationPopupTemp )
      wire#w2
      Contact( #StartConfirmationPopupSel )
      Contact( #StartConfirmationAck )
      wire#w3
      S_Coil( #RMAddStarted )
   END_RUNG
   RUNG wire#w2
      I_Contact( #StartConfirmationPopupSel )
   END_RUNG wire#w3
   RUNG wire#w3
      R_Coil( #StartConfirmationPopupTemp )
   END_RUNG
   RUNG wire#w1
      Contact( #RMAddStarted )
      wire#w4
      Contact( #RMAddAck1 )
      wire#w5
      S_Coil( #RMAddStarted )
   END_RUNG
   RUNG wire#w4
      Contact( #RMAddAck2 )
   END_RUNG wire#w5
   RUNG wire#w4
      Contact( #RMAddAck3 )
   END_RUNG wire#w5
   RUNG wire#w4
      Contact( #RMAddAck4 )
   END_RUNG wire#w5
   RUNG wire#w4
      Contact( #RMAddAck5 )
   END_RUNG wire#w5
   RUNG wire#w4
      Contact( #RMAddAck6 )
   END_RUNG wire#w5
   RUNG wire#w4
      Contact( #RMAddAck7 )
   END_RUNG wire#w5
   RUNG wire#w4
      Contact( #RMAddAck8 )
   END_RUNG wire#w5
   RUNG wire#w4
      Contact( #RMAddAck9 )
   END_RUNG wire#w5
   RUNG wire#w4
      Contact( #RMAddAck10 )
   END_RUNG wire#w5
   RUNG wire#w1
      Contact( #Running )
      wire#w6
      Contact( #StartConfirmationPopupTemp )
      Coil( #StartConfirmationPopup )
   END_RUNG
   RUNG wire#w6
      Contact( #EndConfirmationPopupTemp )
      Coil( #EndConfirmationPopup )
   END_RUNG
   RUNG wire#w6
      Contact( #RMAddStarted )
      Coil( #RMAddPopup )
   END_RUNG
   RUNG wire#w6
      Contact( #DelaytoSettleMaterialPopupTemp )
      Coil( #DelaytoSettleMaterialPopup )
   END_RUNG
   // the same network as SCL:
   #_w1 := #Enable AND #Selected AND NOT #RE2;   // rising edge of #Selected
   #RE2 := #Selected;
   IF #_w1 THEN #StartConfirmationPopupTemp := TRUE; END_IF;
   IF #Enable AND #StartConfirmationPopupTemp AND ((#StartConfirmationPopupSel AND #StartConfirmationAck) OR NOT #StartConfirmationPopupSel) THEN
       #RMAddStarted := TRUE;
       #StartConfirmationPopupTemp := FALSE;
   END_IF;
   IF #Enable AND #RMAddStarted AND (#RMAddAck1 OR #RMAddAck2 OR #RMAddAck3 OR #RMAddAck4 OR #RMAddAck5 OR #RMAddAck6 OR #RMAddAck7 OR #RMAddAck8 OR #RMAddAck9 OR #RMAddAck10) THEN
       #RMAddStarted := TRUE;
   END_IF;
   #_w2 := #Enable AND #Running;
   #StartConfirmationPopup := #_w2 AND #StartConfirmationPopupTemp;
   #EndConfirmationPopup := #_w2 AND #EndConfirmationPopupTemp;
   #RMAddPopup := #_w2 AND #RMAddStarted;
   #DelaytoSettleMaterialPopup := #_w2 AND #DelaytoSettleMaterialPopupTemp;
END_REGION

REGION Network 3: Visibility for RM
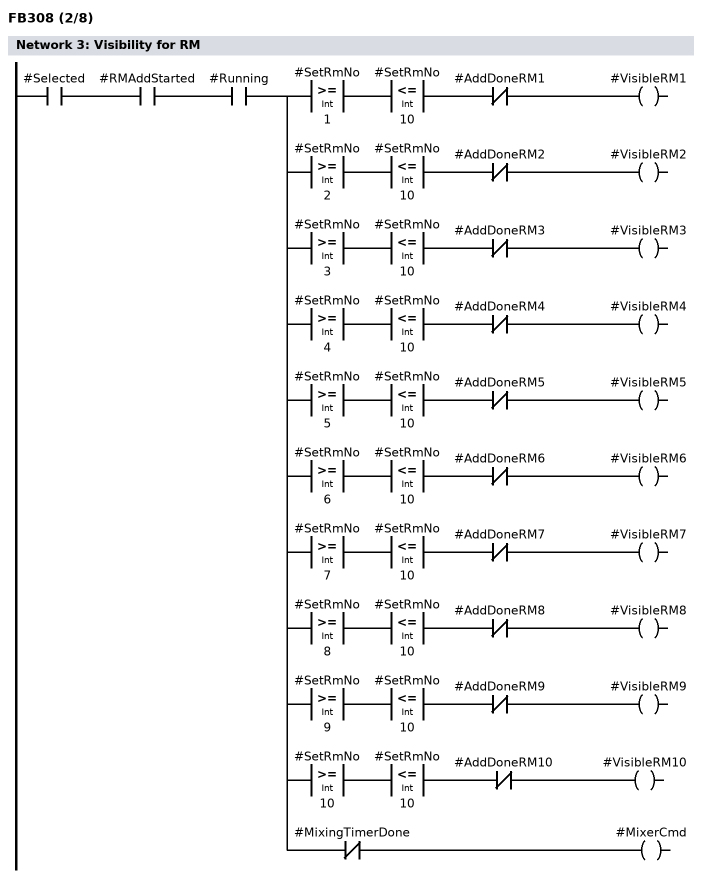
   RUNG wire#powerrail
      Contact( #Selected )
      Contact( #RMAddStarted )
      Contact( #Running )
      wire#w1
      { S7_Templates := "SrcType := Int" } GE_Contact(in1 := #SetRmNo, in2 := 1)
      { S7_Templates := "SrcType := Int" } LE_Contact(in1 := #SetRmNo, in2 := 10)
      I_Contact( #AddDoneRM1 )
      Coil( #VisibleRM1 )
   END_RUNG
   RUNG wire#w1
      { S7_Templates := "SrcType := Int" } GE_Contact(in1 := #SetRmNo, in2 := 2)
      { S7_Templates := "SrcType := Int" } LE_Contact(in1 := #SetRmNo, in2 := 10)
      I_Contact( #AddDoneRM2 )
      Coil( #VisibleRM2 )
   END_RUNG
   RUNG wire#w1
      { S7_Templates := "SrcType := Int" } GE_Contact(in1 := #SetRmNo, in2 := 3)
      { S7_Templates := "SrcType := Int" } LE_Contact(in1 := #SetRmNo, in2 := 10)
      I_Contact( #AddDoneRM3 )
      Coil( #VisibleRM3 )
   END_RUNG
   RUNG wire#w1
      { S7_Templates := "SrcType := Int" } GE_Contact(in1 := #SetRmNo, in2 := 4)
      { S7_Templates := "SrcType := Int" } LE_Contact(in1 := #SetRmNo, in2 := 10)
      I_Contact( #AddDoneRM4 )
      Coil( #VisibleRM4 )
   END_RUNG
   RUNG wire#w1
      { S7_Templates := "SrcType := Int" } GE_Contact(in1 := #SetRmNo, in2 := 5)
      { S7_Templates := "SrcType := Int" } LE_Contact(in1 := #SetRmNo, in2 := 10)
      I_Contact( #AddDoneRM5 )
      Coil( #VisibleRM5 )
   END_RUNG
   RUNG wire#w1
      { S7_Templates := "SrcType := Int" } GE_Contact(in1 := #SetRmNo, in2 := 6)
      { S7_Templates := "SrcType := Int" } LE_Contact(in1 := #SetRmNo, in2 := 10)
      I_Contact( #AddDoneRM6 )
      Coil( #VisibleRM6 )
   END_RUNG
   RUNG wire#w1
      { S7_Templates := "SrcType := Int" } GE_Contact(in1 := #SetRmNo, in2 := 7)
      { S7_Templates := "SrcType := Int" } LE_Contact(in1 := #SetRmNo, in2 := 10)
      I_Contact( #AddDoneRM7 )
      Coil( #VisibleRM7 )
   END_RUNG
   RUNG wire#w1
      { S7_Templates := "SrcType := Int" } GE_Contact(in1 := #SetRmNo, in2 := 8)
      { S7_Templates := "SrcType := Int" } LE_Contact(in1 := #SetRmNo, in2 := 10)
      I_Contact( #AddDoneRM8 )
      Coil( #VisibleRM8 )
   END_RUNG
   RUNG wire#w1
      { S7_Templates := "SrcType := Int" } GE_Contact(in1 := #SetRmNo, in2 := 9)
      { S7_Templates := "SrcType := Int" } LE_Contact(in1 := #SetRmNo, in2 := 10)
      I_Contact( #AddDoneRM9 )
      Coil( #VisibleRM9 )
   END_RUNG
   RUNG wire#w1
      { S7_Templates := "SrcType := Int" } GE_Contact(in1 := #SetRmNo, in2 := 10)
      { S7_Templates := "SrcType := Int" } LE_Contact(in1 := #SetRmNo, in2 := 10)
      I_Contact( #AddDoneRM10 )
      Coil( #VisibleRM10 )
   END_RUNG
   RUNG wire#w1
      I_Contact( #MixingTimerDone )
      Coil( #MixerCmd )
   END_RUNG
   // the same network as SCL:
   #_w1 := #Selected AND #RMAddStarted AND #Running;
   #VisibleRM1 := #_w1 AND (#SetRmNo >= 1) AND (#SetRmNo <= 10) AND NOT #AddDoneRM1;
   #VisibleRM2 := #_w1 AND (#SetRmNo >= 2) AND (#SetRmNo <= 10) AND NOT #AddDoneRM2;
   #VisibleRM3 := #_w1 AND (#SetRmNo >= 3) AND (#SetRmNo <= 10) AND NOT #AddDoneRM3;
   #VisibleRM4 := #_w1 AND (#SetRmNo >= 4) AND (#SetRmNo <= 10) AND NOT #AddDoneRM4;
   #VisibleRM5 := #_w1 AND (#SetRmNo >= 5) AND (#SetRmNo <= 10) AND NOT #AddDoneRM5;
   #VisibleRM6 := #_w1 AND (#SetRmNo >= 6) AND (#SetRmNo <= 10) AND NOT #AddDoneRM6;
   #VisibleRM7 := #_w1 AND (#SetRmNo >= 7) AND (#SetRmNo <= 10) AND NOT #AddDoneRM7;
   #VisibleRM8 := #_w1 AND (#SetRmNo >= 8) AND (#SetRmNo <= 10) AND NOT #AddDoneRM8;
   #VisibleRM9 := #_w1 AND (#SetRmNo >= 9) AND (#SetRmNo <= 10) AND NOT #AddDoneRM9;
   #VisibleRM10 := #_w1 AND (#SetRmNo >= 10) AND (#SetRmNo <= 10) AND NOT #AddDoneRM10;
   #MixerCmd := #_w1 AND NOT #MixingTimerDone;
END_REGION

REGION Network 4: Add Done
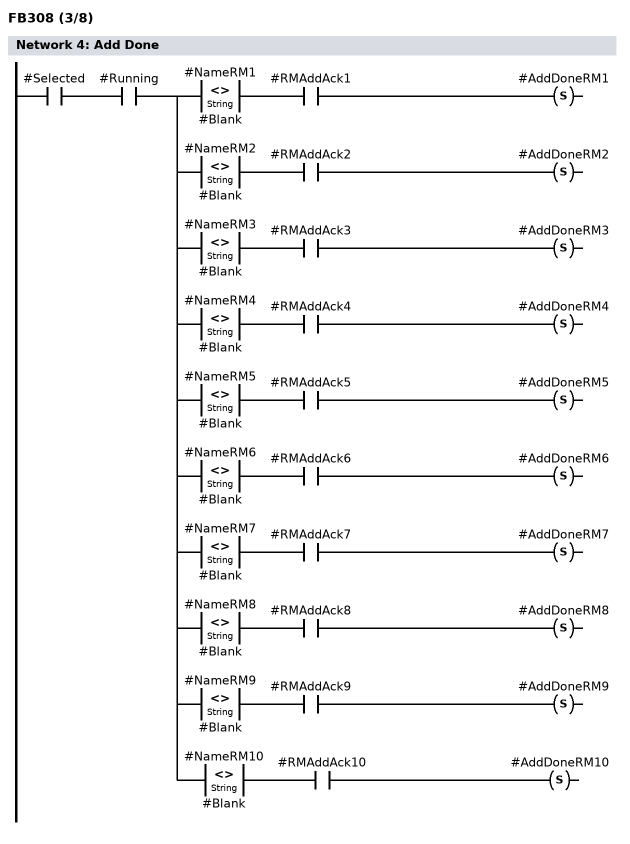
   RUNG wire#powerrail
      Contact( #Selected )
      Contact( #Running )
      wire#w1
      { S7_Templates := "SrcType := String" } NE_Contact(in1 := #NameRM1, in2 := #Blank)
      Contact( #RMAddAck1 )
      S_Coil( #AddDoneRM1 )
   END_RUNG
   RUNG wire#w1
      { S7_Templates := "SrcType := String" } NE_Contact(in1 := #NameRM2, in2 := #Blank)
      Contact( #RMAddAck2 )
      S_Coil( #AddDoneRM2 )
   END_RUNG
   RUNG wire#w1
      { S7_Templates := "SrcType := String" } NE_Contact(in1 := #NameRM3, in2 := #Blank)
      Contact( #RMAddAck3 )
      S_Coil( #AddDoneRM3 )
   END_RUNG
   RUNG wire#w1
      { S7_Templates := "SrcType := String" } NE_Contact(in1 := #NameRM4, in2 := #Blank)
      Contact( #RMAddAck4 )
      S_Coil( #AddDoneRM4 )
   END_RUNG
   RUNG wire#w1
      { S7_Templates := "SrcType := String" } NE_Contact(in1 := #NameRM5, in2 := #Blank)
      Contact( #RMAddAck5 )
      S_Coil( #AddDoneRM5 )
   END_RUNG
   RUNG wire#w1
      { S7_Templates := "SrcType := String" } NE_Contact(in1 := #NameRM6, in2 := #Blank)
      Contact( #RMAddAck6 )
      S_Coil( #AddDoneRM6 )
   END_RUNG
   RUNG wire#w1
      { S7_Templates := "SrcType := String" } NE_Contact(in1 := #NameRM7, in2 := #Blank)
      Contact( #RMAddAck7 )
      S_Coil( #AddDoneRM7 )
   END_RUNG
   RUNG wire#w1
      { S7_Templates := "SrcType := String" } NE_Contact(in1 := #NameRM8, in2 := #Blank)
      Contact( #RMAddAck8 )
      S_Coil( #AddDoneRM8 )
   END_RUNG
   RUNG wire#w1
      { S7_Templates := "SrcType := String" } NE_Contact(in1 := #NameRM9, in2 := #Blank)
      Contact( #RMAddAck9 )
      S_Coil( #AddDoneRM9 )
   END_RUNG
   RUNG wire#w1
      { S7_Templates := "SrcType := String" } NE_Contact(in1 := #NameRM10, in2 := #Blank)
      Contact( #RMAddAck10 )
      S_Coil( #AddDoneRM10 )
   END_RUNG
   // the same network as SCL:
   #_w1 := #Selected AND #Running;
   IF #_w1 AND (#NameRM1 <> #Blank) AND #RMAddAck1 THEN #AddDoneRM1 := TRUE; END_IF;
   IF #_w1 AND (#NameRM2 <> #Blank) AND #RMAddAck2 THEN #AddDoneRM2 := TRUE; END_IF;
   IF #_w1 AND (#NameRM3 <> #Blank) AND #RMAddAck3 THEN #AddDoneRM3 := TRUE; END_IF;
   IF #_w1 AND (#NameRM4 <> #Blank) AND #RMAddAck4 THEN #AddDoneRM4 := TRUE; END_IF;
   IF #_w1 AND (#NameRM5 <> #Blank) AND #RMAddAck5 THEN #AddDoneRM5 := TRUE; END_IF;
   IF #_w1 AND (#NameRM6 <> #Blank) AND #RMAddAck6 THEN #AddDoneRM6 := TRUE; END_IF;
   IF #_w1 AND (#NameRM7 <> #Blank) AND #RMAddAck7 THEN #AddDoneRM7 := TRUE; END_IF;
   IF #_w1 AND (#NameRM8 <> #Blank) AND #RMAddAck8 THEN #AddDoneRM8 := TRUE; END_IF;
   IF #_w1 AND (#NameRM9 <> #Blank) AND #RMAddAck9 THEN #AddDoneRM9 := TRUE; END_IF;
   IF #_w1 AND (#NameRM10 <> #Blank) AND #RMAddAck10 THEN #AddDoneRM10 := TRUE; END_IF;
END_REGION

REGION Network 5: All Addition Done
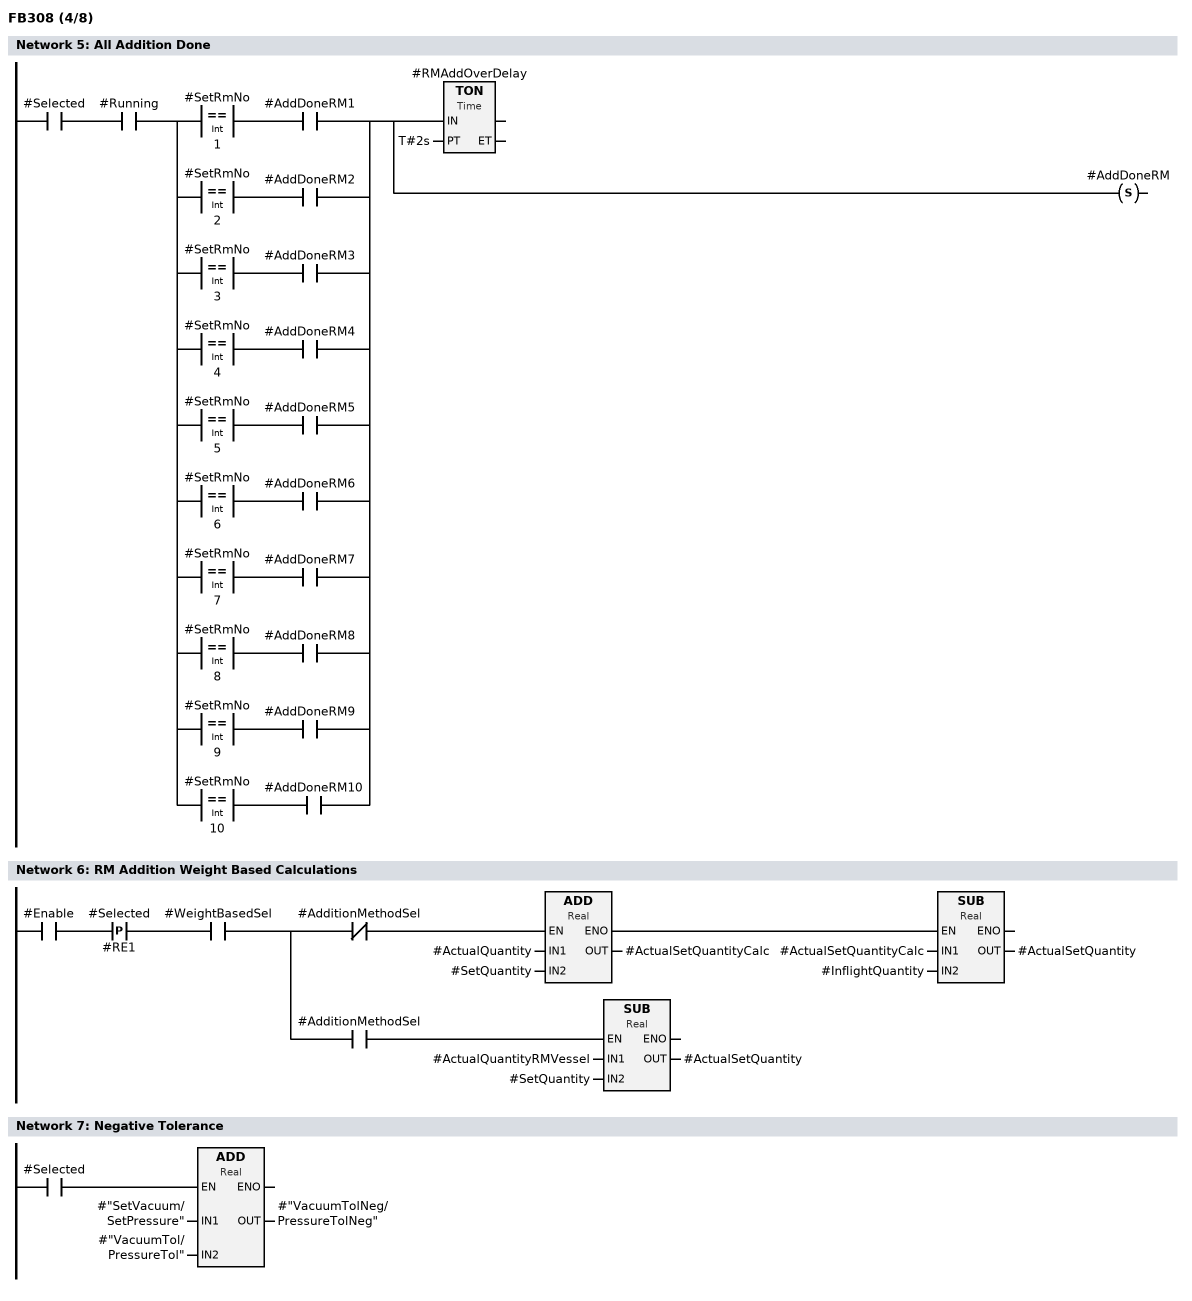
   RUNG wire#powerrail
      Contact( #Selected )
      Contact( #Running )
      wire#w1
      { S7_Templates := "SrcType := Int" } EQ_Contact(in1 := #SetRmNo, in2 := 1)
      Contact( #AddDoneRM1 )
      wire#w2
      { S7_Templates := "time_type := Time" } #RMAddOverDelay.TON(pt := T#2s, et =>)
   END_RUNG
   RUNG wire#w1
      { S7_Templates := "SrcType := Int" } EQ_Contact(in1 := #SetRmNo, in2 := 2)
      Contact( #AddDoneRM2 )
   END_RUNG wire#w2
   RUNG wire#w1
      { S7_Templates := "SrcType := Int" } EQ_Contact(in1 := #SetRmNo, in2 := 3)
      Contact( #AddDoneRM3 )
   END_RUNG wire#w2
   RUNG wire#w1
      { S7_Templates := "SrcType := Int" } EQ_Contact(in1 := #SetRmNo, in2 := 4)
      Contact( #AddDoneRM4 )
   END_RUNG wire#w2
   RUNG wire#w1
      { S7_Templates := "SrcType := Int" } EQ_Contact(in1 := #SetRmNo, in2 := 5)
      Contact( #AddDoneRM5 )
   END_RUNG wire#w2
   RUNG wire#w1
      { S7_Templates := "SrcType := Int" } EQ_Contact(in1 := #SetRmNo, in2 := 6)
      Contact( #AddDoneRM6 )
   END_RUNG wire#w2
   RUNG wire#w1
      { S7_Templates := "SrcType := Int" } EQ_Contact(in1 := #SetRmNo, in2 := 7)
      Contact( #AddDoneRM7 )
   END_RUNG wire#w2
   RUNG wire#w1
      { S7_Templates := "SrcType := Int" } EQ_Contact(in1 := #SetRmNo, in2 := 8)
      Contact( #AddDoneRM8 )
   END_RUNG wire#w2
   RUNG wire#w1
      { S7_Templates := "SrcType := Int" } EQ_Contact(in1 := #SetRmNo, in2 := 9)
      Contact( #AddDoneRM9 )
   END_RUNG wire#w2
   RUNG wire#w1
      { S7_Templates := "SrcType := Int" } EQ_Contact(in1 := #SetRmNo, in2 := 10)
      Contact( #AddDoneRM10 )
   END_RUNG wire#w2
   RUNG wire#w2
      S_Coil( #AddDoneRM )
   END_RUNG
   // the same network as SCL:
   #_w1 := #Selected AND #Running AND (((#SetRmNo = 1) AND #AddDoneRM1) OR ((#SetRmNo = 2) AND #AddDoneRM2) OR ((#SetRmNo = 3) AND #AddDoneRM3) OR ((#SetRmNo = 4) AND #AddDoneRM4) OR ((#SetRmNo = 5) AND #AddDoneRM5) OR ((#SetRmNo = 6) AND #AddDoneRM6) OR ((#SetRmNo = 7) AND #AddDoneRM7) OR ((#SetRmNo = 8) AND #AddDoneRM8) OR ((#SetRmNo = 9) AND #AddDoneRM9) OR ((#SetRmNo = 10) AND #AddDoneRM10));
   #RMAddOverDelay(IN := #_w1, PT := T#2s);   // TON
   IF #_w1 THEN #AddDoneRM := TRUE; END_IF;
END_REGION

REGION Network 6: RM Addition Weight Based Calculations
   RUNG wire#powerrail
      Contact( #Enable )
      P_Contact(operand := #Selected, bit := #RE1)
      Contact( #WeightBasedSel )
      wire#w1
      I_Contact( #AdditionMethodSel )
      { S7_Templates := "SrcType := Real"; S7_GenerateENO := "TRUE" } Add(in1 := #ActualQuantity, in2 := #SetQuantity, out => #ActualSetQuantityCalc)
      { S7_Templates := "SrcType := Real"; S7_GenerateENO := "TRUE" } Sub(in1 := #ActualSetQuantityCalc, in2 := #InflightQuantity, out => #ActualSetQuantity)
   END_RUNG
   RUNG wire#w1
      Contact( #AdditionMethodSel )
      { S7_Templates := "SrcType := Real"; S7_GenerateENO := "TRUE" } Sub(in1 := #ActualQuantityRMVessel, in2 := #SetQuantity, out => #ActualSetQuantity)
   END_RUNG
   // the same network as SCL:
   // ENO of a box is taken as its EN; it also drops when the box reports an error
   #_w1 := #Enable AND #Selected AND NOT #RE1;   // rising edge of #Selected
   #RE1 := #Selected;
   #_w2 := #_w1 AND #WeightBasedSel;
   IF #_w2 AND NOT #AdditionMethodSel THEN
       #ActualSetQuantityCalc := #ActualQuantity + #SetQuantity;
       #ActualSetQuantity := #ActualSetQuantityCalc - #InflightQuantity;
   END_IF;
   IF #_w2 AND #AdditionMethodSel THEN #ActualSetQuantity := #ActualQuantityRMVessel - #SetQuantity; END_IF;
END_REGION

REGION Network 7: Negative Tolerance
   RUNG wire#powerrail
      Contact( #Selected )
      { S7_Templates := "SrcType := Real"; S7_GenerateENO := "TRUE" } Add(in1 := #"SetVacuum/SetPressure", in2 := #"VacuumTol/PressureTol", out => #"VacuumTolNeg/PressureTolNeg")
   END_RUNG
   // the same network as SCL:
   IF #Selected THEN
       #"VacuumTolNeg/PressureTolNeg" := #"SetVacuum/SetPressure" + #"VacuumTol/PressureTol";
   END_IF;
END_REGION

REGION Network 8: Outputs
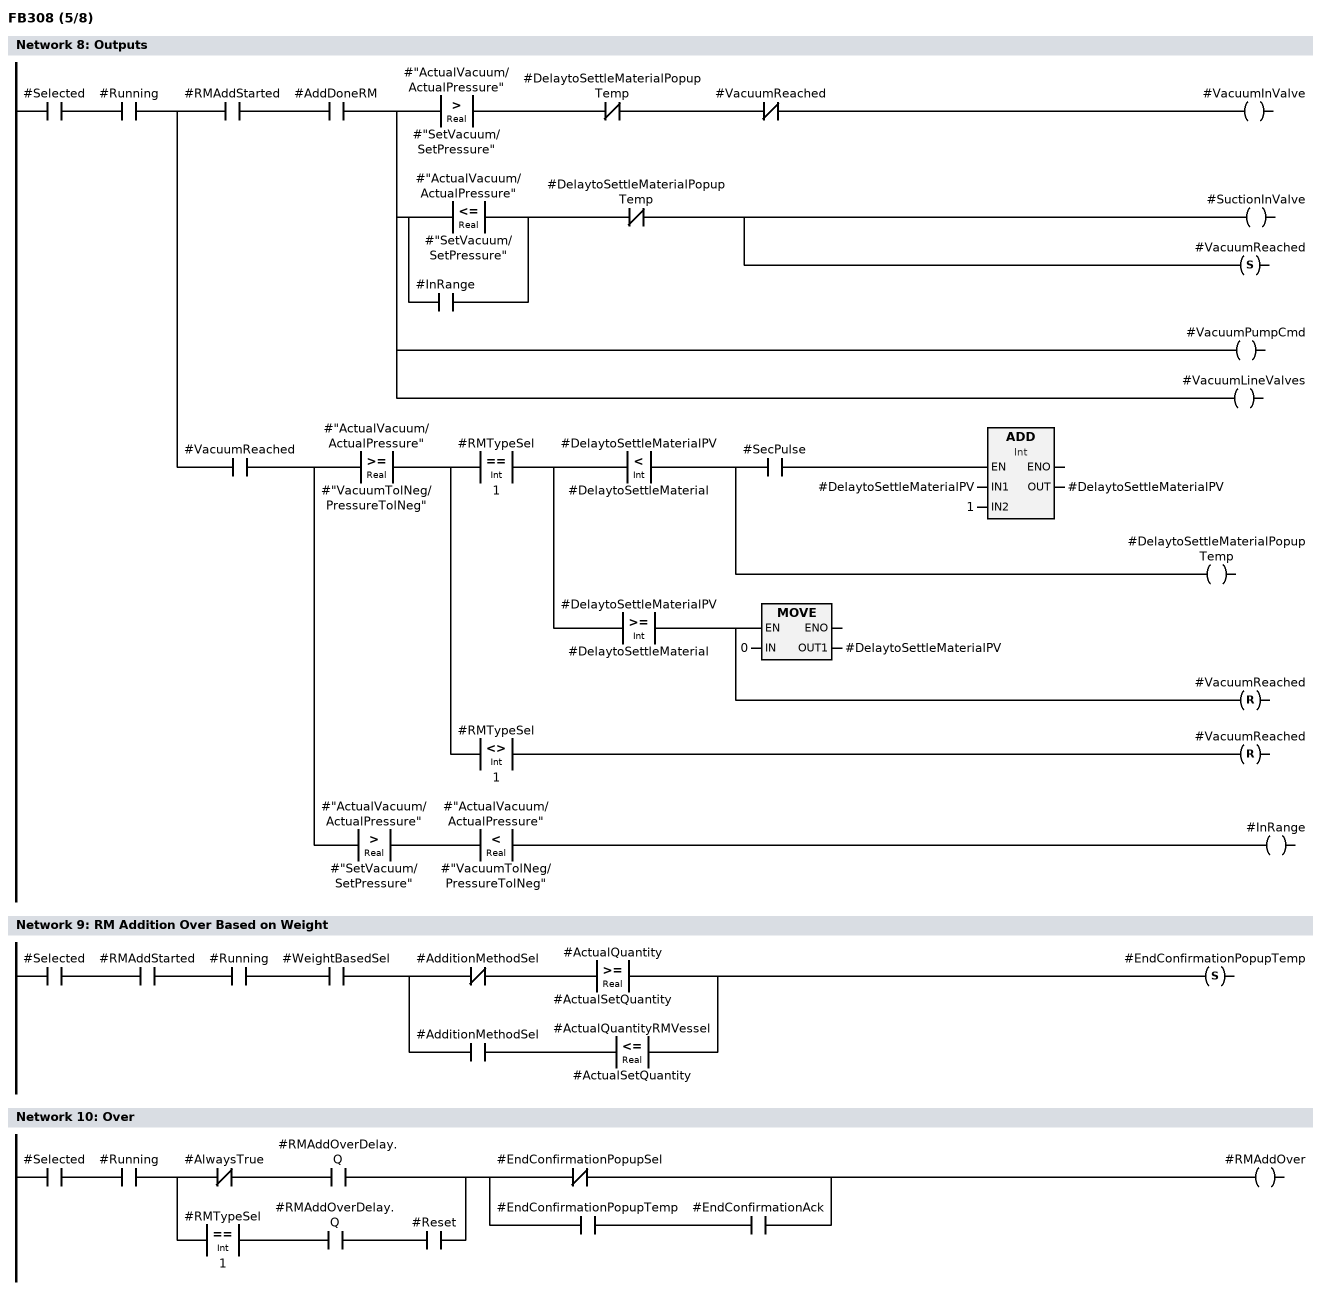
   RUNG wire#powerrail
      Contact( #Selected )
      Contact( #Running )
      wire#w1
      Contact( #RMAddStarted )
      Contact( #AddDoneRM )
      wire#w2
      { S7_Templates := "SrcType := Real" } GT_Contact(in1 := #"ActualVacuum/ActualPressure", in2 := #"SetVacuum/SetPressure")
      I_Contact( #DelaytoSettleMaterialPopupTemp )
      I_Contact( #VacuumReached )
      Coil( #VacuumInValve )
   END_RUNG
   RUNG wire#w2
      { S7_Templates := "SrcType := Real" } LE_Contact(in1 := #"ActualVacuum/ActualPressure", in2 := #"SetVacuum/SetPressure")
      wire#w3
      I_Contact( #DelaytoSettleMaterialPopupTemp )
      wire#w4
      Coil( #SuctionInValve )
   END_RUNG
   RUNG wire#w2
      Contact( #InRange )
   END_RUNG wire#w3
   RUNG wire#w4
      S_Coil( #VacuumReached )
   END_RUNG
   RUNG wire#w2
      Coil( #VacuumPumpCmd )
   END_RUNG
   RUNG wire#w2
      Coil( #VacuumLineValves )
   END_RUNG
   RUNG wire#w1
      Contact( #VacuumReached )
      wire#w5
      { S7_Templates := "SrcType := Real" } GE_Contact(in1 := #"ActualVacuum/ActualPressure", in2 := #"VacuumTolNeg/PressureTolNeg")
      wire#w6
      { S7_Templates := "SrcType := Int" } EQ_Contact(in1 := #RMTypeSel, in2 := 1)
      wire#w7
      { S7_Templates := "SrcType := Int" } LT_Contact(in1 := #DelaytoSettleMaterialPV, in2 := #DelaytoSettleMaterial)
      wire#w8
      Contact( #SecPulse )
      { S7_Templates := "SrcType := Int"; S7_GenerateENO := "TRUE" } Add(in1 := #DelaytoSettleMaterialPV, in2 := 1, out => #DelaytoSettleMaterialPV)
   END_RUNG
   RUNG wire#w8
      Coil( #DelaytoSettleMaterialPopupTemp )
   END_RUNG
   RUNG wire#w7
      { S7_Templates := "SrcType := Int" } GE_Contact(in1 := #DelaytoSettleMaterialPV, in2 := #DelaytoSettleMaterial)
      wire#w9
      { S7_GenerateENO := "TRUE" } Move(in := 0, out1 => #DelaytoSettleMaterialPV)
   END_RUNG
   RUNG wire#w9
      R_Coil( #VacuumReached )
   END_RUNG
   RUNG wire#w6
      { S7_Templates := "SrcType := Int" } NE_Contact(in1 := #RMTypeSel, in2 := 1)
      R_Coil( #VacuumReached )
   END_RUNG
   RUNG wire#w5
      { S7_Templates := "SrcType := Real" } GT_Contact(in1 := #"ActualVacuum/ActualPressure", in2 := #"SetVacuum/SetPressure")
      { S7_Templates := "SrcType := Real" } LT_Contact(in1 := #"ActualVacuum/ActualPressure", in2 := #"VacuumTolNeg/PressureTolNeg")
      Coil( #InRange )
   END_RUNG
   // the same network as SCL:
   #_w1 := #Selected AND #Running;
   #_w2 := #_w1 AND #RMAddStarted AND #AddDoneRM;
   #VacuumInValve := #_w2 AND (#"ActualVacuum/ActualPressure" > #"SetVacuum/SetPressure") AND NOT #DelaytoSettleMaterialPopupTemp AND NOT #VacuumReached;
   #SuctionInValve := #_w2 AND ((#"ActualVacuum/ActualPressure" <= #"SetVacuum/SetPressure") OR #InRange) AND NOT #DelaytoSettleMaterialPopupTemp;
   IF #SuctionInValve THEN #VacuumReached := TRUE; END_IF;
   #VacuumPumpCmd := #_w2;
   #VacuumLineValves := #_w2;
   #_w3 := #_w1 AND #VacuumReached;
   #_w4 := #_w3 AND (#"ActualVacuum/ActualPressure" >= #"VacuumTolNeg/PressureTolNeg");
   #_w5 := #_w4 AND (#RMTypeSel = 1);
   #_w6 := #_w5 AND (#DelaytoSettleMaterialPV < #DelaytoSettleMaterial);
   IF #_w6 AND #SecPulse THEN #DelaytoSettleMaterialPV := #DelaytoSettleMaterialPV + 1; END_IF;
   #DelaytoSettleMaterialPopupTemp := #_w6;
   #_w7 := #_w5 AND (#DelaytoSettleMaterialPV >= #DelaytoSettleMaterial);
   IF #_w7 THEN
       #DelaytoSettleMaterialPV := 0;
       #VacuumReached := FALSE;
   END_IF;
   IF #_w4 AND (#RMTypeSel <> 1) THEN #VacuumReached := FALSE; END_IF;
   #InRange := #_w3 AND (#"ActualVacuum/ActualPressure" > #"SetVacuum/SetPressure") AND (#"ActualVacuum/ActualPressure" < #"VacuumTolNeg/PressureTolNeg");
END_REGION

REGION Network 9: RM Addition Over Based on Weight
   RUNG wire#powerrail
      Contact( #Selected )
      Contact( #RMAddStarted )
      Contact( #Running )
      Contact( #WeightBasedSel )
      wire#w1
      I_Contact( #AdditionMethodSel )
      { S7_Templates := "SrcType := Real" } GE_Contact(in1 := #ActualQuantity, in2 := #ActualSetQuantity)
      wire#w2
      S_Coil( #EndConfirmationPopupTemp )
   END_RUNG
   RUNG wire#w1
      Contact( #AdditionMethodSel )
      { S7_Templates := "SrcType := Real" } LE_Contact(in1 := #ActualQuantityRMVessel, in2 := #ActualSetQuantity)
   END_RUNG wire#w2
   // the same network as SCL:
   IF #Selected AND #RMAddStarted AND #Running AND #WeightBasedSel AND ((NOT #AdditionMethodSel AND (#ActualQuantity >= #ActualSetQuantity)) OR (#AdditionMethodSel AND (#ActualQuantityRMVessel <= #ActualSetQuantity))) THEN
       #EndConfirmationPopupTemp := TRUE;
   END_IF;
END_REGION

REGION Network 10: Over
   RUNG wire#powerrail
      Contact( #Selected )
      Contact( #Running )
      wire#w1
      I_Contact( #AlwaysTrue )
      Contact( #RMAddOverDelay.Q )
      wire#w2
      I_Contact( #EndConfirmationPopupSel )
      wire#w3
      Coil( #RMAddOver )
   END_RUNG
   RUNG wire#w1
      { S7_Templates := "SrcType := Int" } EQ_Contact(in1 := #RMTypeSel, in2 := 1)
      Contact( #RMAddOverDelay.Q )
      Contact( #Reset )
   END_RUNG wire#w2
   RUNG wire#w2
      Contact( #EndConfirmationPopupTemp )
      Contact( #EndConfirmationAck )
   END_RUNG wire#w3
   // the same network as SCL:
   #RMAddOver := #Selected AND #Running AND ((NOT #AlwaysTrue AND #RMAddOverDelay.Q) OR ((#RMTypeSel = 1) AND #RMAddOverDelay.Q AND #Reset)) AND (NOT #EndConfirmationPopupSel OR (#EndConfirmationPopupTemp AND #EndConfirmationAck));
END_REGION

REGION Network 11: Event Status
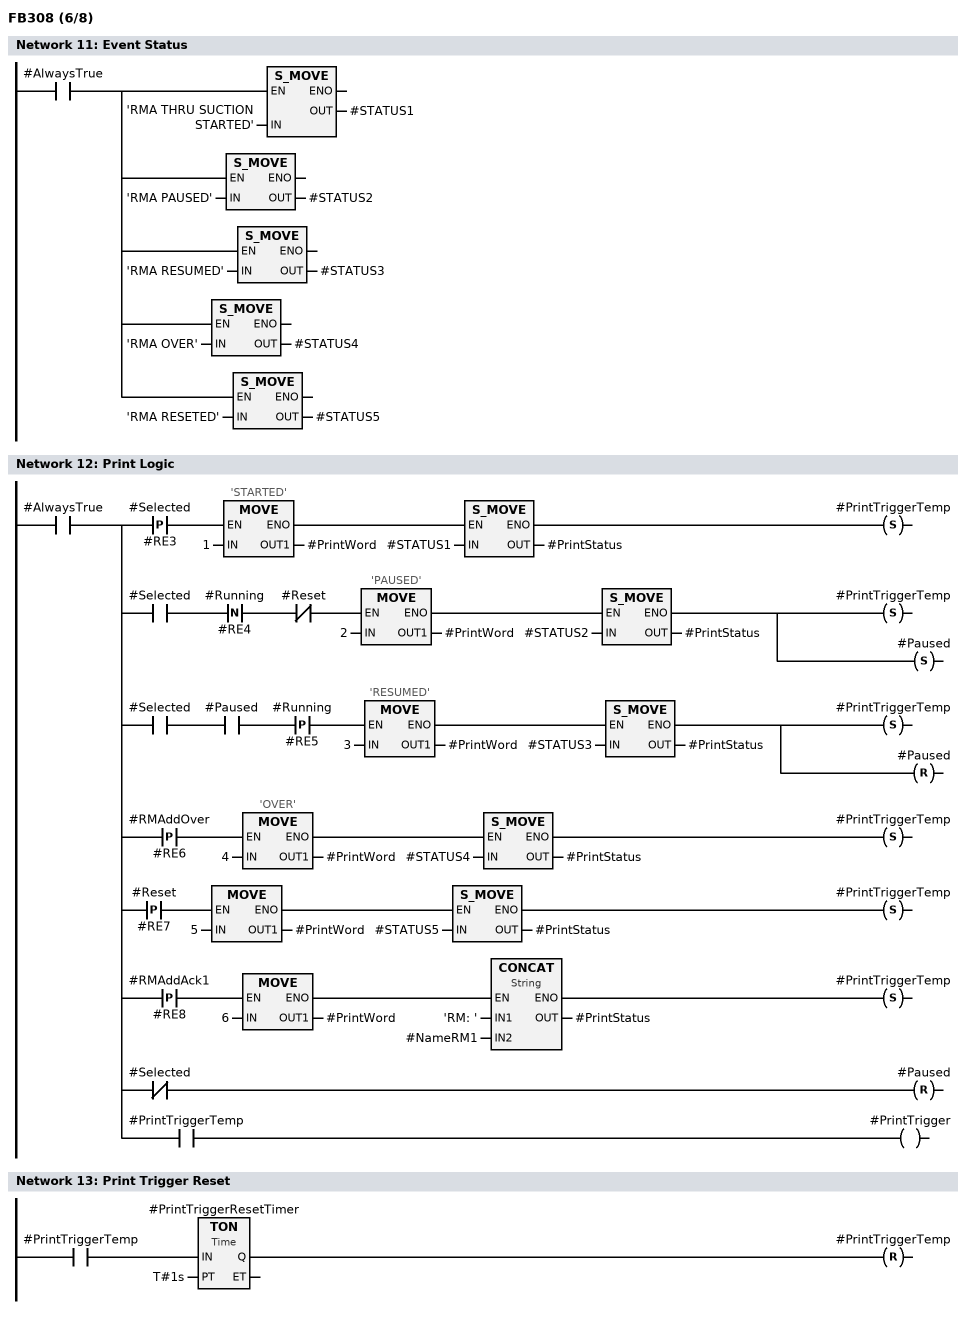
   RUNG wire#powerrail
      Contact( #AlwaysTrue )
      wire#w1
      S_Move(in := 'RMA THRU SUCTION STARTED', out => #STATUS1)
   END_RUNG
   RUNG wire#w1
      S_Move(in := 'RMA PAUSED', out => #STATUS2)
   END_RUNG
   RUNG wire#w1
      S_Move(in := 'RMA RESUMED', out => #STATUS3)
   END_RUNG
   RUNG wire#w1
      S_Move(in := 'RMA OVER', out => #STATUS4)
   END_RUNG
   RUNG wire#w1
      S_Move(in := 'RMA RESETED', out => #STATUS5)
   END_RUNG
   // the same network as SCL:
   IF #AlwaysTrue THEN
       #STATUS1 := 'RMA THRU SUCTION STARTED';
       #STATUS2 := 'RMA PAUSED';
       #STATUS3 := 'RMA RESUMED';
       #STATUS4 := 'RMA OVER';
       #STATUS5 := 'RMA RESETED';
   END_IF;
END_REGION

REGION Network 12: Print Logic
   RUNG wire#powerrail
      Contact( #AlwaysTrue )
      wire#w1
      P_Contact(operand := #Selected, bit := #RE3)
      { S7_GenerateENO := "TRUE" } Move(in := 1, out1 => #PrintWord)   // 'STARTED'
      S_Move(in := #STATUS1, out => #PrintStatus)
      S_Coil( #PrintTriggerTemp )
   END_RUNG
   RUNG wire#w1
      Contact( #Selected )
      N_Contact(operand := #Running, bit := #RE4)
      I_Contact( #Reset )
      { S7_GenerateENO := "TRUE" } Move(in := 2, out1 => #PrintWord)   // 'PAUSED'
      S_Move(in := #STATUS2, out => #PrintStatus)
      wire#w2
      S_Coil( #PrintTriggerTemp )
   END_RUNG
   RUNG wire#w2
      S_Coil( #Paused )
   END_RUNG
   RUNG wire#w1
      Contact( #Selected )
      Contact( #Paused )
      P_Contact(operand := #Running, bit := #RE5)
      { S7_GenerateENO := "TRUE" } Move(in := 3, out1 => #PrintWord)   // 'RESUMED'
      S_Move(in := #STATUS3, out => #PrintStatus)
      wire#w3
      S_Coil( #PrintTriggerTemp )
   END_RUNG
   RUNG wire#w3
      R_Coil( #Paused )
   END_RUNG
   RUNG wire#w1
      P_Contact(operand := #RMAddOver, bit := #RE6)
      { S7_GenerateENO := "TRUE" } Move(in := 4, out1 => #PrintWord)   // 'OVER'
      S_Move(in := #STATUS4, out => #PrintStatus)
      S_Coil( #PrintTriggerTemp )
   END_RUNG
   RUNG wire#w1
      P_Contact(operand := #Reset, bit := #RE7)
      { S7_GenerateENO := "TRUE" } Move(in := 5, out1 => #PrintWord)
      S_Move(in := #STATUS5, out => #PrintStatus)
      S_Coil( #PrintTriggerTemp )
   END_RUNG
   RUNG wire#w1
      P_Contact(operand := #RMAddAck1, bit := #RE8)
      { S7_GenerateENO := "TRUE" } Move(in := 6, out1 => #PrintWord)
      { S7_Templates := "[card := 2, str_type := String]" } CONCAT(IN1 := 'RM: ', IN2 := #NameRM1, OUT => #PrintStatus)
      S_Coil( #PrintTriggerTemp )
   END_RUNG
   RUNG wire#w1
      I_Contact( #Selected )
      R_Coil( #Paused )
   END_RUNG
   RUNG wire#w1
      Contact( #PrintTriggerTemp )
      Coil( #PrintTrigger )
   END_RUNG
   // the same network as SCL:
   // ENO of a box is taken as its EN; it also drops when the box reports an error
   #_w1 := #AlwaysTrue AND #Selected AND NOT #RE3;   // rising edge of #Selected
   #RE3 := #Selected;
   IF #_w1 THEN
       #PrintWord := 1;   // 'STARTED'
       #PrintStatus := #STATUS1;
       #PrintTriggerTemp := TRUE;
   END_IF;
   #_w2 := #AlwaysTrue AND #Selected AND NOT #Running AND #RE4;   // falling edge of #Running
   #RE4 := #Running;
   IF #_w2 AND NOT #Reset THEN
       #PrintWord := 2;   // 'PAUSED'
       #PrintStatus := #STATUS2;
       #PrintTriggerTemp := TRUE;
       #Paused := TRUE;
   END_IF;
   #_w3 := #AlwaysTrue AND #Selected AND #Paused AND #Running AND NOT #RE5;   // rising edge of #Running
   #RE5 := #Running;
   IF #_w3 THEN
       #PrintWord := 3;   // 'RESUMED'
       #PrintStatus := #STATUS3;
       #PrintTriggerTemp := TRUE;
       #Paused := FALSE;
   END_IF;
   #_w4 := #AlwaysTrue AND #RMAddOver AND NOT #RE6;   // rising edge of #RMAddOver
   #RE6 := #RMAddOver;
   IF #_w4 THEN
       #PrintWord := 4;   // 'OVER'
       #PrintStatus := #STATUS4;
       #PrintTriggerTemp := TRUE;
   END_IF;
   #_w5 := #AlwaysTrue AND #Reset AND NOT #RE7;   // rising edge of #Reset
   #RE7 := #Reset;
   IF #_w5 THEN
       #PrintWord := 5;
       #PrintStatus := #STATUS5;
       #PrintTriggerTemp := TRUE;
   END_IF;
   #_w6 := #AlwaysTrue AND #RMAddAck1 AND NOT #RE8;   // rising edge of #RMAddAck1
   #RE8 := #RMAddAck1;
   IF #_w6 THEN #PrintWord := 6; END_IF;
   CONCAT(EN := #_w6, IN1 := 'RM: ', IN2 := #NameRM1, OUT => #PrintStatus, ENO => #_w7);
   IF #_w7 THEN #PrintTriggerTemp := TRUE; END_IF;
   IF #AlwaysTrue AND NOT #Selected THEN #Paused := FALSE; END_IF;
   #PrintTrigger := #AlwaysTrue AND #PrintTriggerTemp;
END_REGION

REGION Network 13: Print Trigger Reset
   RUNG wire#powerrail
      Contact( #PrintTriggerTemp )
      { S7_Templates := "time_type := Time" } #PrintTriggerResetTimer.TON(pt := T#1s, et =>)
      R_Coil( #PrintTriggerTemp )
   END_RUNG
   // the same network as SCL:
   #PrintTriggerResetTimer(IN := #PrintTriggerTemp, PT := T#1s);   // TON
   IF #PrintTriggerResetTimer.Q THEN #PrintTriggerTemp := FALSE; END_IF;
END_REGION

REGION Network 14: Button Reset
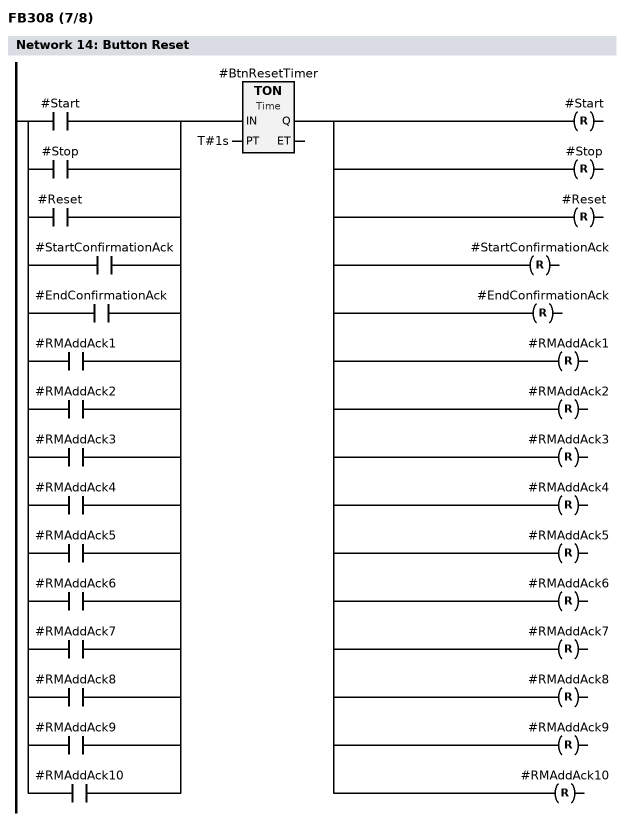
   RUNG wire#powerrail
      Contact( #Start )
      wire#w1
      { S7_Templates := "time_type := Time" } #BtnResetTimer.TON(pt := T#1s, et =>)
      wire#w2
      R_Coil( #Start )
   END_RUNG
   RUNG wire#powerrail
      Contact( #Stop )
   END_RUNG wire#w1
   RUNG wire#powerrail
      Contact( #Reset )
   END_RUNG wire#w1
   RUNG wire#powerrail
      Contact( #StartConfirmationAck )
   END_RUNG wire#w1
   RUNG wire#powerrail
      Contact( #EndConfirmationAck )
   END_RUNG wire#w1
   RUNG wire#powerrail
      Contact( #RMAddAck1 )
   END_RUNG wire#w1
   RUNG wire#powerrail
      Contact( #RMAddAck2 )
   END_RUNG wire#w1
   RUNG wire#powerrail
      Contact( #RMAddAck3 )
   END_RUNG wire#w1
   RUNG wire#powerrail
      Contact( #RMAddAck4 )
   END_RUNG wire#w1
   RUNG wire#powerrail
      Contact( #RMAddAck5 )
   END_RUNG wire#w1
   RUNG wire#powerrail
      Contact( #RMAddAck6 )
   END_RUNG wire#w1
   RUNG wire#powerrail
      Contact( #RMAddAck7 )
   END_RUNG wire#w1
   RUNG wire#powerrail
      Contact( #RMAddAck8 )
   END_RUNG wire#w1
   RUNG wire#powerrail
      Contact( #RMAddAck9 )
   END_RUNG wire#w1
   RUNG wire#powerrail
      Contact( #RMAddAck10 )
   END_RUNG wire#w1
   RUNG wire#w2
      R_Coil( #Stop )
   END_RUNG
   RUNG wire#w2
      R_Coil( #Reset )
   END_RUNG
   RUNG wire#w2
      R_Coil( #StartConfirmationAck )
   END_RUNG
   RUNG wire#w2
      R_Coil( #EndConfirmationAck )
   END_RUNG
   RUNG wire#w2
      R_Coil( #RMAddAck1 )
   END_RUNG
   RUNG wire#w2
      R_Coil( #RMAddAck2 )
   END_RUNG
   RUNG wire#w2
      R_Coil( #RMAddAck3 )
   END_RUNG
   RUNG wire#w2
      R_Coil( #RMAddAck4 )
   END_RUNG
   RUNG wire#w2
      R_Coil( #RMAddAck5 )
   END_RUNG
   RUNG wire#w2
      R_Coil( #RMAddAck6 )
   END_RUNG
   RUNG wire#w2
      R_Coil( #RMAddAck7 )
   END_RUNG
   RUNG wire#w2
      R_Coil( #RMAddAck8 )
   END_RUNG
   RUNG wire#w2
      R_Coil( #RMAddAck9 )
   END_RUNG
   RUNG wire#w2
      R_Coil( #RMAddAck10 )
   END_RUNG
   // the same network as SCL:
   #BtnResetTimer(IN := #Start OR #Stop OR #Reset OR #StartConfirmationAck OR #EndConfirmationAck OR #RMAddAck1 OR #RMAddAck2 OR #RMAddAck3 OR #RMAddAck4 OR #RMAddAck5 OR #RMAddAck6 OR #RMAddAck7 OR #RMAddAck8 OR #RMAddAck9 OR #RMAddAck10,   // TON
                  PT := T#1s);
   IF #BtnResetTimer.Q THEN
       #Start := FALSE;
       #Stop := FALSE;
       #Reset := FALSE;
       #StartConfirmationAck := FALSE;
       #EndConfirmationAck := FALSE;
       #RMAddAck1 := FALSE;
       #RMAddAck2 := FALSE;
       #RMAddAck3 := FALSE;
       #RMAddAck4 := FALSE;
       #RMAddAck5 := FALSE;
       #RMAddAck6 := FALSE;
       #RMAddAck7 := FALSE;
       #RMAddAck8 := FALSE;
       #RMAddAck9 := FALSE;
       #RMAddAck10 := FALSE;
   END_IF;
END_REGION

REGION Network 15: Reset
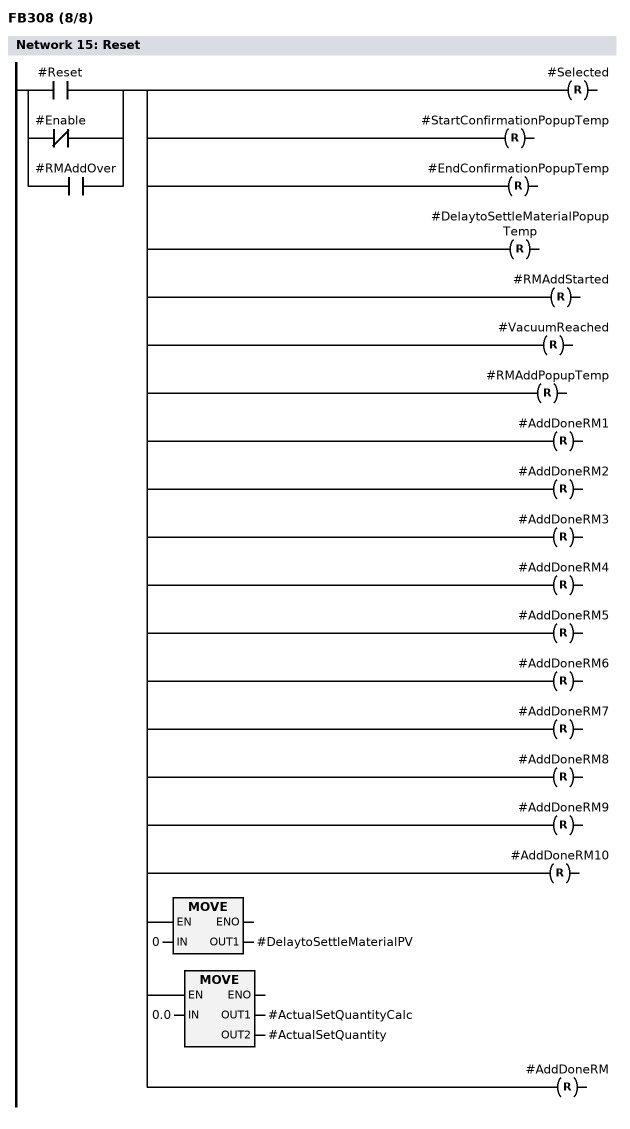
   RUNG wire#powerrail
      Contact( #Reset )
      wire#w1
      R_Coil( #Selected )
   END_RUNG
   RUNG wire#powerrail
      I_Contact( #Enable )
   END_RUNG wire#w1
   RUNG wire#powerrail
      Contact( #RMAddOver )
   END_RUNG wire#w1
   RUNG wire#w1
      R_Coil( #StartConfirmationPopupTemp )
   END_RUNG
   RUNG wire#w1
      R_Coil( #EndConfirmationPopupTemp )
   END_RUNG
   RUNG wire#w1
      R_Coil( #DelaytoSettleMaterialPopupTemp )
   END_RUNG
   RUNG wire#w1
      R_Coil( #RMAddStarted )
   END_RUNG
   RUNG wire#w1
      R_Coil( #VacuumReached )
   END_RUNG
   RUNG wire#w1
      R_Coil( #RMAddPopupTemp )
   END_RUNG
   RUNG wire#w1
      R_Coil( #AddDoneRM1 )
   END_RUNG
   RUNG wire#w1
      R_Coil( #AddDoneRM2 )
   END_RUNG
   RUNG wire#w1
      R_Coil( #AddDoneRM3 )
   END_RUNG
   RUNG wire#w1
      R_Coil( #AddDoneRM4 )
   END_RUNG
   RUNG wire#w1
      R_Coil( #AddDoneRM5 )
   END_RUNG
   RUNG wire#w1
      R_Coil( #AddDoneRM6 )
   END_RUNG
   RUNG wire#w1
      R_Coil( #AddDoneRM7 )
   END_RUNG
   RUNG wire#w1
      R_Coil( #AddDoneRM8 )
   END_RUNG
   RUNG wire#w1
      R_Coil( #AddDoneRM9 )
   END_RUNG
   RUNG wire#w1
      R_Coil( #AddDoneRM10 )
   END_RUNG
   RUNG wire#w1
      Move(in := 0, out1 => #DelaytoSettleMaterialPV)
   END_RUNG
   RUNG wire#w1
      Move(in := 0.0, out1 => #ActualSetQuantityCalc, out2 => #ActualSetQuantity)
   END_RUNG
   RUNG wire#w1
      R_Coil( #AddDoneRM )
   END_RUNG
   // the same network as SCL:
   IF #Reset OR NOT #Enable OR #RMAddOver THEN
       #Selected := FALSE;
       #StartConfirmationPopupTemp := FALSE;
       #EndConfirmationPopupTemp := FALSE;
       #DelaytoSettleMaterialPopupTemp := FALSE;
       #RMAddStarted := FALSE;
       #VacuumReached := FALSE;
       #RMAddPopupTemp := FALSE;
       #AddDoneRM1 := FALSE;
       #AddDoneRM2 := FALSE;
       #AddDoneRM3 := FALSE;
       #AddDoneRM4 := FALSE;
       #AddDoneRM5 := FALSE;
       #AddDoneRM6 := FALSE;
       #AddDoneRM7 := FALSE;
       #AddDoneRM8 := FALSE;
       #AddDoneRM9 := FALSE;
       #AddDoneRM10 := FALSE;
       #DelaytoSettleMaterialPV := 0;
       #ActualSetQuantityCalc := 0.0;
       #ActualSetQuantity := 0.0;
       #AddDoneRM := FALSE;
   END_IF;
END_REGION
END_FUNCTION_BLOCK

FUNCTION_BLOCK "FB309"   // FB309, LAD
TITLE = FB309
{ S7_Optimized_Access := 'FALSE' }
AUTHOR : PRECISE
FAMILY : PRECISE
// RAW MATERIAL ADDITION LIQUID DRUM
// stored: AutoNumber false, SetENOAutomatically false
   VAR_INPUT
      Enable : Bool;
      Disable : Bool;
      Fault : Bool;
      SecPulse : Bool;
      AlwaysTrue : Bool;
      StartConfirmationPopupSel : Bool;   // StartConfirmationPopupSel: 0-NO/1-YES
      EndConfirmationPopupSel : Bool;   // EndConfirmationPopupSel: 0-NO/1-YES
      WeightBasedSel : Bool;   // Weight Based Sel: 0-NO/1-YES
      AdditionMethodSel : Bool;   // Addition Method : 0-Add In Weight/1-Loss In Weight
      RMAddPopupSel : Bool;   // RM Add Popup Sel: 0-NO/1-YES
      SetQuantity : Real := 10.0;   // Weight Based Sel: 1-YES
      SetSpeed : Real := 50.0;
      ActualQuantity : Real;   // Collecting Vessel Weight
      ActualQuantityRMVessel : Real;   // Transffering Vessel Weight
      InflightQuantity : Real;
      DelaytoStartPump : Int := 3;
   END_VAR
   VAR_OUTPUT
      LineValves : Bool;
      PumpCmd : Bool;
      StartConfirmationPopup : Bool;   // For Start Confirmation Popup Selection: Yes
      EndConfirmationPopup : Bool;   // For End Confirmation Popup Selection: Yes
      RMAddPopup : Bool;   // For RMAddPopupSel: 1-YES
      ActualSpeed : Real;
      PrintTrigger : Bool;
      PrintWord : Int;
      PrintStatus : String[50];
   END_VAR
   VAR_IN_OUT
      Start : Bool;
      Stop : Bool;
      Reset : Bool;
      StartConfirmationAck : Bool;   // For Start Confirmation Popup Selection: Yes
      EndConfirmationAck : Bool;   // For End Confirmation Popup Selection: Yes
      RMAddAck : Bool;   // For RMAddPopupSel: 1-YES
      SpareBtn1 : Bool;
      SpareBtn2 : Bool;
      Running : Bool;
      Selected : Bool;
      Paused : Bool;
      StartConfirmationPopupTemp : Bool;   // For Start Confirmation Popup Selection: Yes
      EndConfirmationPopupTemp : Bool;   // For End Confirmation Popup Selection: Yes
      RMAddPopupTemp : Bool;   // For RMAddPopupSel: 1-YES
      RMAddStarted : Bool;
      RMAddOver : Bool;
      ActualSetQuantityCalc : Real;   // For WeightBaseSel: 1-YES
      ActualSetQuantity : Real;   // For WeightBaseSel: 1-YES
   END_VAR
   VAR
      ValveOnDelayPV : Int;
      ValveOffDelayPV : Int;
      PrintTriggerTemp : Bool;
      RE1 : Bool;
      RE2 : Bool;
      RE3 : Bool;
      RE4 : Bool;
      RE5 : Bool;
      RE6 : Bool;
      RE7 : Bool;
      RE8 : Bool;
      PrintTriggerResetTimer { S7_SetPoint := 'True'} : TON_TIME;
      BtnResetTimer { S7_SetPoint := 'True'} : TON_TIME;
      NameRM : String[40];
   END_VAR
   VAR_TEMP
      STATUS1 : String[40];
      STATUS2 : String[40];
      STATUS3 : String[40];
      STATUS4 : String[40];
      STATUS5 : String[40];
   END_VAR
   VAR_TEMP   // added for the SCL form of the ladder/FBD networks
      _w1 : Bool;
      _w2 : Bool;
      _w3 : Bool;
      _w4 : Bool;
      _w5 : Bool;
      _w6 : Bool;
      _w7 : Bool;
   END_VAR
BEGIN

REGION Network 1: Running
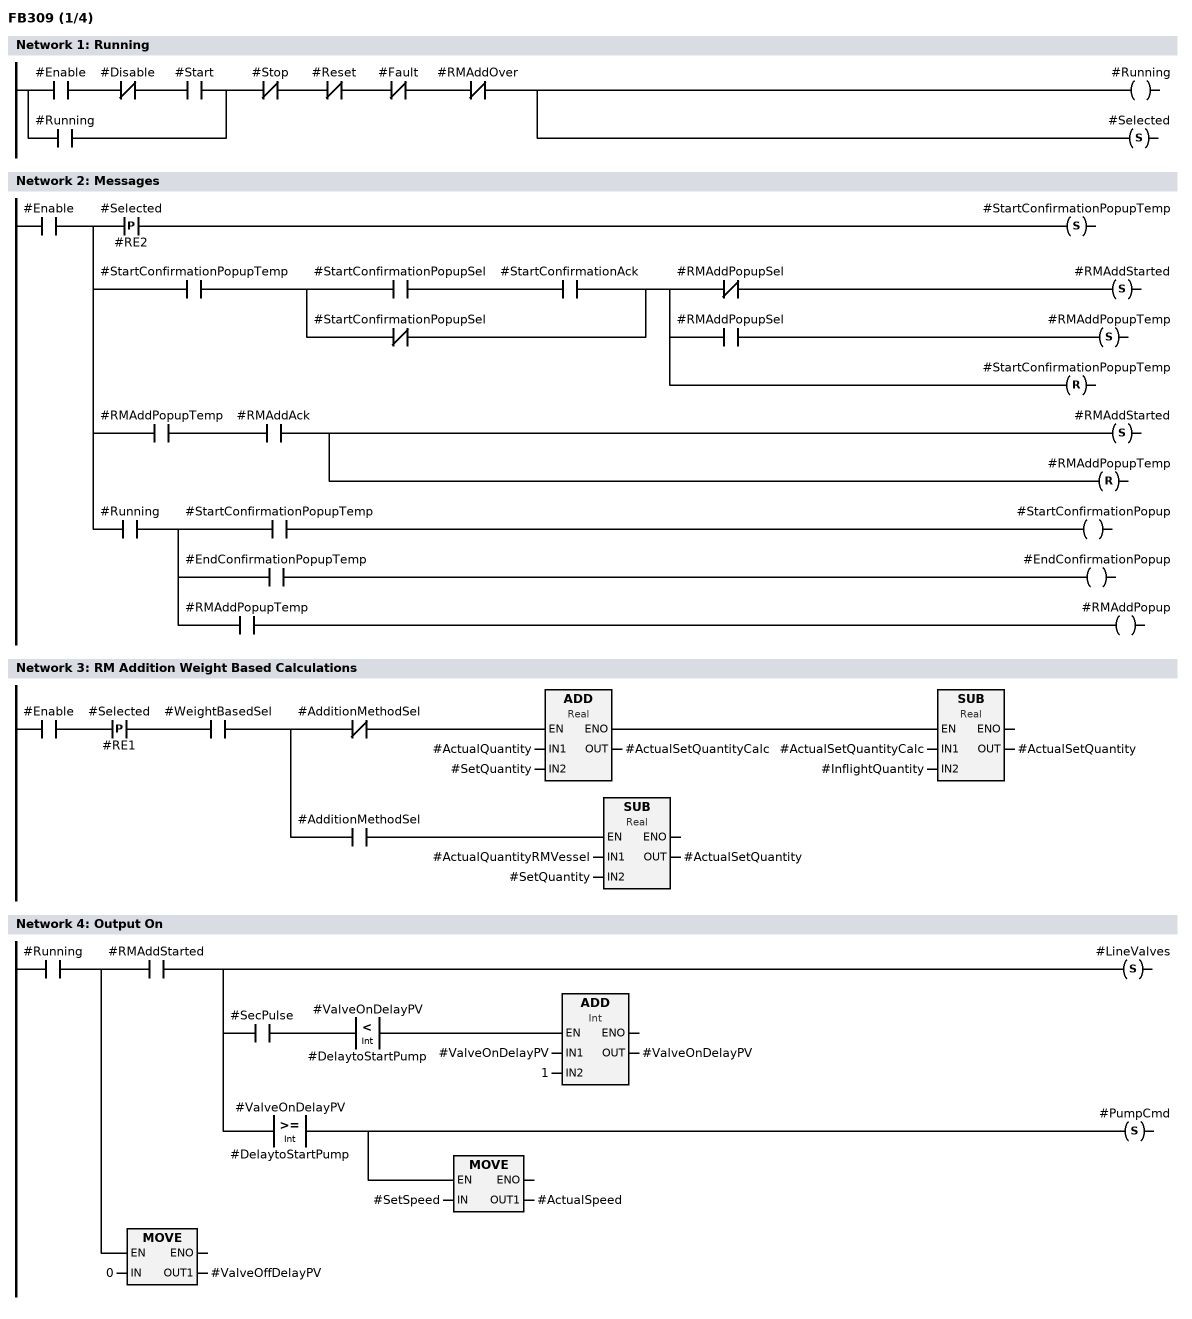
   RUNG wire#powerrail
      Contact( #Enable )
      I_Contact( #Disable )
      Contact( #Start )
      wire#w1
      I_Contact( #Stop )
      I_Contact( #Reset )
      I_Contact( #Fault )
      I_Contact( #RMAddOver )
      wire#w2
      Coil( #Running )
   END_RUNG
   RUNG wire#powerrail
      Contact( #Running )
   END_RUNG wire#w1
   RUNG wire#w2
      S_Coil( #Selected )
   END_RUNG
   // the same network as SCL:
   #Running := ((#Enable AND NOT #Disable AND #Start) OR #Running) AND NOT #Stop AND NOT #Reset AND NOT #Fault AND NOT #RMAddOver;
   IF #Running THEN #Selected := TRUE; END_IF;
END_REGION

REGION Network 2: Messages
   RUNG wire#powerrail
      Contact( #Enable )
      wire#w1
      P_Contact(operand := #Selected, bit := #RE2)
      S_Coil( #StartConfirmationPopupTemp )
   END_RUNG
   RUNG wire#w1
      Contact( #StartConfirmationPopupTemp )
      wire#w2
      Contact( #StartConfirmationPopupSel )
      Contact( #StartConfirmationAck )
      wire#w3
      I_Contact( #RMAddPopupSel )
      S_Coil( #RMAddStarted )
   END_RUNG
   RUNG wire#w2
      I_Contact( #StartConfirmationPopupSel )
   END_RUNG wire#w3
   RUNG wire#w3
      Contact( #RMAddPopupSel )
      S_Coil( #RMAddPopupTemp )
   END_RUNG
   RUNG wire#w3
      R_Coil( #StartConfirmationPopupTemp )
   END_RUNG
   RUNG wire#w1
      Contact( #RMAddPopupTemp )
      Contact( #RMAddAck )
      wire#w4
      S_Coil( #RMAddStarted )
   END_RUNG
   RUNG wire#w4
      R_Coil( #RMAddPopupTemp )
   END_RUNG
   RUNG wire#w1
      Contact( #Running )
      wire#w5
      Contact( #StartConfirmationPopupTemp )
      Coil( #StartConfirmationPopup )
   END_RUNG
   RUNG wire#w5
      Contact( #EndConfirmationPopupTemp )
      Coil( #EndConfirmationPopup )
   END_RUNG
   RUNG wire#w5
      Contact( #RMAddPopupTemp )
      Coil( #RMAddPopup )
   END_RUNG
   // the same network as SCL:
   #_w1 := #Enable AND #Selected AND NOT #RE2;   // rising edge of #Selected
   #RE2 := #Selected;
   IF #_w1 THEN #StartConfirmationPopupTemp := TRUE; END_IF;
   #_w2 := #Enable AND #StartConfirmationPopupTemp AND ((#StartConfirmationPopupSel AND #StartConfirmationAck) OR NOT #StartConfirmationPopupSel);
   IF #_w2 AND NOT #RMAddPopupSel THEN #RMAddStarted := TRUE; END_IF;
   IF #_w2 AND #RMAddPopupSel THEN #RMAddPopupTemp := TRUE; END_IF;
   IF #_w2 THEN #StartConfirmationPopupTemp := FALSE; END_IF;
   IF #Enable AND #RMAddPopupTemp AND #RMAddAck THEN
       #RMAddStarted := TRUE;
       #RMAddPopupTemp := FALSE;
   END_IF;
   #_w3 := #Enable AND #Running;
   #StartConfirmationPopup := #_w3 AND #StartConfirmationPopupTemp;
   #EndConfirmationPopup := #_w3 AND #EndConfirmationPopupTemp;
   #RMAddPopup := #_w3 AND #RMAddPopupTemp;
END_REGION

REGION Network 3: RM Addition Weight Based Calculations
   RUNG wire#powerrail
      Contact( #Enable )
      P_Contact(operand := #Selected, bit := #RE1)
      Contact( #WeightBasedSel )
      wire#w1
      I_Contact( #AdditionMethodSel )
      { S7_Templates := "SrcType := Real"; S7_GenerateENO := "TRUE" } Add(in1 := #ActualQuantity, in2 := #SetQuantity, out => #ActualSetQuantityCalc)
      { S7_Templates := "SrcType := Real"; S7_GenerateENO := "TRUE" } Sub(in1 := #ActualSetQuantityCalc, in2 := #InflightQuantity, out => #ActualSetQuantity)
   END_RUNG
   RUNG wire#w1
      Contact( #AdditionMethodSel )
      { S7_Templates := "SrcType := Real"; S7_GenerateENO := "TRUE" } Sub(in1 := #ActualQuantityRMVessel, in2 := #SetQuantity, out => #ActualSetQuantity)
   END_RUNG
   // the same network as SCL:
   // ENO of a box is taken as its EN; it also drops when the box reports an error
   #_w1 := #Enable AND #Selected AND NOT #RE1;   // rising edge of #Selected
   #RE1 := #Selected;
   #_w2 := #_w1 AND #WeightBasedSel;
   IF #_w2 AND NOT #AdditionMethodSel THEN
       #ActualSetQuantityCalc := #ActualQuantity + #SetQuantity;
       #ActualSetQuantity := #ActualSetQuantityCalc - #InflightQuantity;
   END_IF;
   IF #_w2 AND #AdditionMethodSel THEN #ActualSetQuantity := #ActualQuantityRMVessel - #SetQuantity; END_IF;
END_REGION

REGION Network 4: Output On
   RUNG wire#powerrail
      Contact( #Running )
      wire#w1
      Contact( #RMAddStarted )
      wire#w2
      S_Coil( #LineValves )
   END_RUNG
   RUNG wire#w2
      Contact( #SecPulse )
      { S7_Templates := "SrcType := Int" } LT_Contact(in1 := #ValveOnDelayPV, in2 := #DelaytoStartPump)
      { S7_Templates := "SrcType := Int"; S7_GenerateENO := "TRUE" } Add(in1 := #ValveOnDelayPV, in2 := 1, out => #ValveOnDelayPV)
   END_RUNG
   RUNG wire#w2
      { S7_Templates := "SrcType := Int" } GE_Contact(in1 := #ValveOnDelayPV, in2 := #DelaytoStartPump)
      wire#w3
      S_Coil( #PumpCmd )
   END_RUNG
   RUNG wire#w3
      Move(in := #SetSpeed, out1 => #ActualSpeed)
   END_RUNG
   RUNG wire#w1
      { S7_GenerateENO := "TRUE" } Move(in := 0, out1 => #ValveOffDelayPV)
   END_RUNG
   // the same network as SCL:
   #_w1 := #Running AND #RMAddStarted;
   IF #_w1 THEN #LineValves := TRUE; END_IF;
   IF #_w1 AND #SecPulse AND (#ValveOnDelayPV < #DelaytoStartPump) THEN
       #ValveOnDelayPV := #ValveOnDelayPV + 1;
   END_IF;
   IF #_w1 AND (#ValveOnDelayPV >= #DelaytoStartPump) THEN
       #PumpCmd := TRUE;
       #ActualSpeed := #SetSpeed;
   END_IF;
   IF #Running THEN #ValveOffDelayPV := 0; END_IF;
END_REGION

REGION Network 5: Output Off
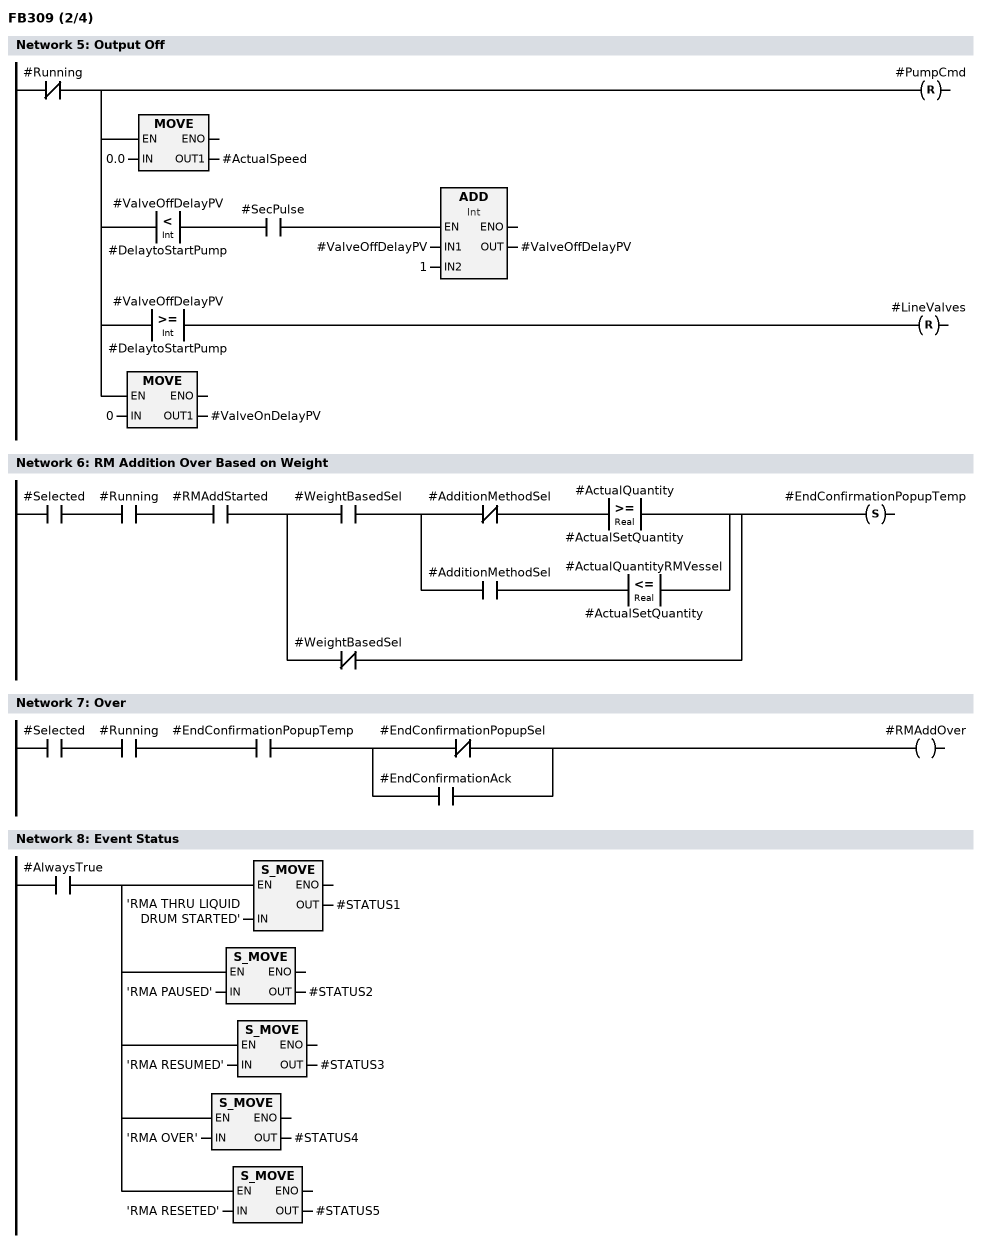
   RUNG wire#powerrail
      I_Contact( #Running )
      wire#w1
      R_Coil( #PumpCmd )
   END_RUNG
   RUNG wire#w1
      Move(in := 0.0, out1 => #ActualSpeed)
   END_RUNG
   RUNG wire#w1
      { S7_Templates := "SrcType := Int" } LT_Contact(in1 := #ValveOffDelayPV, in2 := #DelaytoStartPump)
      Contact( #SecPulse )
      { S7_Templates := "SrcType := Int"; S7_GenerateENO := "TRUE" } Add(in1 := #ValveOffDelayPV, in2 := 1, out => #ValveOffDelayPV)
   END_RUNG
   RUNG wire#w1
      { S7_Templates := "SrcType := Int" } GE_Contact(in1 := #ValveOffDelayPV, in2 := #DelaytoStartPump)
      R_Coil( #LineValves )
   END_RUNG
   RUNG wire#w1
      { S7_GenerateENO := "TRUE" } Move(in := 0, out1 => #ValveOnDelayPV)
   END_RUNG
   // the same network as SCL:
   IF NOT #Running THEN
       #PumpCmd := FALSE;
       #ActualSpeed := 0.0;
   END_IF;
   IF NOT #Running AND (#ValveOffDelayPV < #DelaytoStartPump) AND #SecPulse THEN
       #ValveOffDelayPV := #ValveOffDelayPV + 1;
   END_IF;
   IF NOT #Running AND (#ValveOffDelayPV >= #DelaytoStartPump) THEN #LineValves := FALSE; END_IF;
   IF NOT #Running THEN #ValveOnDelayPV := 0; END_IF;
END_REGION

REGION Network 6: RM Addition Over Based on Weight
   RUNG wire#powerrail
      Contact( #Selected )
      Contact( #Running )
      Contact( #RMAddStarted )
      wire#w1
      Contact( #WeightBasedSel )
      wire#w2
      I_Contact( #AdditionMethodSel )
      { S7_Templates := "SrcType := Real" } GE_Contact(in1 := #ActualQuantity, in2 := #ActualSetQuantity)
      wire#w3
      S_Coil( #EndConfirmationPopupTemp )
   END_RUNG
   RUNG wire#w2
      Contact( #AdditionMethodSel )
      { S7_Templates := "SrcType := Real" } LE_Contact(in1 := #ActualQuantityRMVessel, in2 := #ActualSetQuantity)
   END_RUNG wire#w3
   RUNG wire#w1
      I_Contact( #WeightBasedSel )
   END_RUNG wire#w3
   // the same network as SCL:
   IF #Selected AND #Running AND #RMAddStarted AND ((#WeightBasedSel AND ((NOT #AdditionMethodSel AND (#ActualQuantity >= #ActualSetQuantity)) OR (#AdditionMethodSel AND (#ActualQuantityRMVessel <= #ActualSetQuantity)))) OR NOT #WeightBasedSel) THEN
       #EndConfirmationPopupTemp := TRUE;
   END_IF;
END_REGION

REGION Network 7: Over
   RUNG wire#powerrail
      Contact( #Selected )
      Contact( #Running )
      Contact( #EndConfirmationPopupTemp )
      wire#w1
      I_Contact( #EndConfirmationPopupSel )
      wire#w2
      Coil( #RMAddOver )
   END_RUNG
   RUNG wire#w1
      Contact( #EndConfirmationAck )
   END_RUNG wire#w2
   // the same network as SCL:
   #RMAddOver := #Selected AND #Running AND #EndConfirmationPopupTemp AND (NOT #EndConfirmationPopupSel OR #EndConfirmationAck);
END_REGION

REGION Network 8: Event Status
   RUNG wire#powerrail
      Contact( #AlwaysTrue )
      wire#w1
      S_Move(in := 'RMA THRU LIQUID DRUM STARTED', out => #STATUS1)
   END_RUNG
   RUNG wire#w1
      S_Move(in := 'RMA PAUSED', out => #STATUS2)
   END_RUNG
   RUNG wire#w1
      S_Move(in := 'RMA RESUMED', out => #STATUS3)
   END_RUNG
   RUNG wire#w1
      S_Move(in := 'RMA OVER', out => #STATUS4)
   END_RUNG
   RUNG wire#w1
      S_Move(in := 'RMA RESETED', out => #STATUS5)
   END_RUNG
   // the same network as SCL:
   IF #AlwaysTrue THEN
       #STATUS1 := 'RMA THRU LIQUID DRUM STARTED';
       #STATUS2 := 'RMA PAUSED';
       #STATUS3 := 'RMA RESUMED';
       #STATUS4 := 'RMA OVER';
       #STATUS5 := 'RMA RESETED';
   END_IF;
END_REGION

REGION Network 9: Print Logic
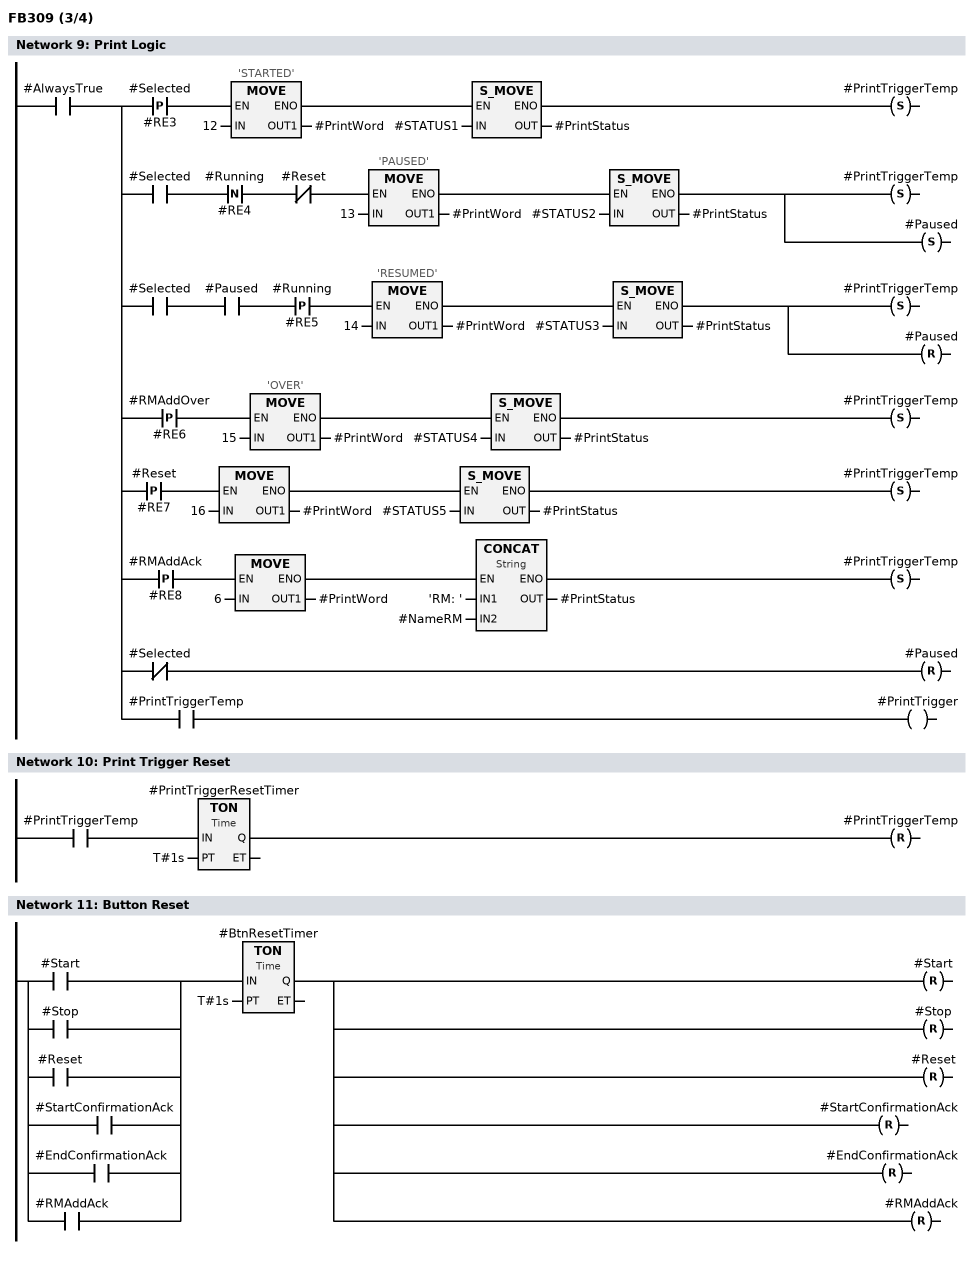
   RUNG wire#powerrail
      Contact( #AlwaysTrue )
      wire#w1
      P_Contact(operand := #Selected, bit := #RE3)
      { S7_GenerateENO := "TRUE" } Move(in := 12, out1 => #PrintWord)   // 'STARTED'
      S_Move(in := #STATUS1, out => #PrintStatus)
      S_Coil( #PrintTriggerTemp )
   END_RUNG
   RUNG wire#w1
      Contact( #Selected )
      N_Contact(operand := #Running, bit := #RE4)
      I_Contact( #Reset )
      { S7_GenerateENO := "TRUE" } Move(in := 13, out1 => #PrintWord)   // 'PAUSED'
      S_Move(in := #STATUS2, out => #PrintStatus)
      wire#w2
      S_Coil( #PrintTriggerTemp )
   END_RUNG
   RUNG wire#w2
      S_Coil( #Paused )
   END_RUNG
   RUNG wire#w1
      Contact( #Selected )
      Contact( #Paused )
      P_Contact(operand := #Running, bit := #RE5)
      { S7_GenerateENO := "TRUE" } Move(in := 14, out1 => #PrintWord)   // 'RESUMED'
      S_Move(in := #STATUS3, out => #PrintStatus)
      wire#w3
      S_Coil( #PrintTriggerTemp )
   END_RUNG
   RUNG wire#w3
      R_Coil( #Paused )
   END_RUNG
   RUNG wire#w1
      P_Contact(operand := #RMAddOver, bit := #RE6)
      { S7_GenerateENO := "TRUE" } Move(in := 15, out1 => #PrintWord)   // 'OVER'
      S_Move(in := #STATUS4, out => #PrintStatus)
      S_Coil( #PrintTriggerTemp )
   END_RUNG
   RUNG wire#w1
      P_Contact(operand := #Reset, bit := #RE7)
      { S7_GenerateENO := "TRUE" } Move(in := 16, out1 => #PrintWord)
      S_Move(in := #STATUS5, out => #PrintStatus)
      S_Coil( #PrintTriggerTemp )
   END_RUNG
   RUNG wire#w1
      P_Contact(operand := #RMAddAck, bit := #RE8)
      { S7_GenerateENO := "TRUE" } Move(in := 6, out1 => #PrintWord)
      { S7_Templates := "[card := 2, str_type := String]" } CONCAT(IN1 := 'RM: ', IN2 := #NameRM, OUT => #PrintStatus)
      S_Coil( #PrintTriggerTemp )
   END_RUNG
   RUNG wire#w1
      I_Contact( #Selected )
      R_Coil( #Paused )
   END_RUNG
   RUNG wire#w1
      Contact( #PrintTriggerTemp )
      Coil( #PrintTrigger )
   END_RUNG
   // the same network as SCL:
   // ENO of a box is taken as its EN; it also drops when the box reports an error
   #_w1 := #AlwaysTrue AND #Selected AND NOT #RE3;   // rising edge of #Selected
   #RE3 := #Selected;
   IF #_w1 THEN
       #PrintWord := 12;   // 'STARTED'
       #PrintStatus := #STATUS1;
       #PrintTriggerTemp := TRUE;
   END_IF;
   #_w2 := #AlwaysTrue AND #Selected AND NOT #Running AND #RE4;   // falling edge of #Running
   #RE4 := #Running;
   IF #_w2 AND NOT #Reset THEN
       #PrintWord := 13;   // 'PAUSED'
       #PrintStatus := #STATUS2;
       #PrintTriggerTemp := TRUE;
       #Paused := TRUE;
   END_IF;
   #_w3 := #AlwaysTrue AND #Selected AND #Paused AND #Running AND NOT #RE5;   // rising edge of #Running
   #RE5 := #Running;
   IF #_w3 THEN
       #PrintWord := 14;   // 'RESUMED'
       #PrintStatus := #STATUS3;
       #PrintTriggerTemp := TRUE;
       #Paused := FALSE;
   END_IF;
   #_w4 := #AlwaysTrue AND #RMAddOver AND NOT #RE6;   // rising edge of #RMAddOver
   #RE6 := #RMAddOver;
   IF #_w4 THEN
       #PrintWord := 15;   // 'OVER'
       #PrintStatus := #STATUS4;
       #PrintTriggerTemp := TRUE;
   END_IF;
   #_w5 := #AlwaysTrue AND #Reset AND NOT #RE7;   // rising edge of #Reset
   #RE7 := #Reset;
   IF #_w5 THEN
       #PrintWord := 16;
       #PrintStatus := #STATUS5;
       #PrintTriggerTemp := TRUE;
   END_IF;
   #_w6 := #AlwaysTrue AND #RMAddAck AND NOT #RE8;   // rising edge of #RMAddAck
   #RE8 := #RMAddAck;
   IF #_w6 THEN #PrintWord := 6; END_IF;
   CONCAT(EN := #_w6, IN1 := 'RM: ', IN2 := #NameRM, OUT => #PrintStatus, ENO => #_w7);
   IF #_w7 THEN #PrintTriggerTemp := TRUE; END_IF;
   IF #AlwaysTrue AND NOT #Selected THEN #Paused := FALSE; END_IF;
   #PrintTrigger := #AlwaysTrue AND #PrintTriggerTemp;
END_REGION

REGION Network 10: Print Trigger Reset
   RUNG wire#powerrail
      Contact( #PrintTriggerTemp )
      { S7_Templates := "time_type := Time" } #PrintTriggerResetTimer.TON(pt := T#1s, et =>)
      R_Coil( #PrintTriggerTemp )
   END_RUNG
   // the same network as SCL:
   #PrintTriggerResetTimer(IN := #PrintTriggerTemp, PT := T#1s);   // TON
   IF #PrintTriggerResetTimer.Q THEN #PrintTriggerTemp := FALSE; END_IF;
END_REGION

REGION Network 11: Button Reset
   RUNG wire#powerrail
      Contact( #Start )
      wire#w1
      { S7_Templates := "time_type := Time" } #BtnResetTimer.TON(pt := T#1s, et =>)
      wire#w2
      R_Coil( #Start )
   END_RUNG
   RUNG wire#powerrail
      Contact( #Stop )
   END_RUNG wire#w1
   RUNG wire#powerrail
      Contact( #Reset )
   END_RUNG wire#w1
   RUNG wire#powerrail
      Contact( #StartConfirmationAck )
   END_RUNG wire#w1
   RUNG wire#powerrail
      Contact( #EndConfirmationAck )
   END_RUNG wire#w1
   RUNG wire#powerrail
      Contact( #RMAddAck )
   END_RUNG wire#w1
   RUNG wire#w2
      R_Coil( #Stop )
   END_RUNG
   RUNG wire#w2
      R_Coil( #Reset )
   END_RUNG
   RUNG wire#w2
      R_Coil( #StartConfirmationAck )
   END_RUNG
   RUNG wire#w2
      R_Coil( #EndConfirmationAck )
   END_RUNG
   RUNG wire#w2
      R_Coil( #RMAddAck )
   END_RUNG
   // the same network as SCL:
   #BtnResetTimer(IN := #Start OR #Stop OR #Reset OR #StartConfirmationAck OR #EndConfirmationAck OR #RMAddAck,   // TON
                  PT := T#1s);
   IF #BtnResetTimer.Q THEN
       #Start := FALSE;
       #Stop := FALSE;
       #Reset := FALSE;
       #StartConfirmationAck := FALSE;
       #EndConfirmationAck := FALSE;
       #RMAddAck := FALSE;
   END_IF;
END_REGION

REGION Network 12: Reset
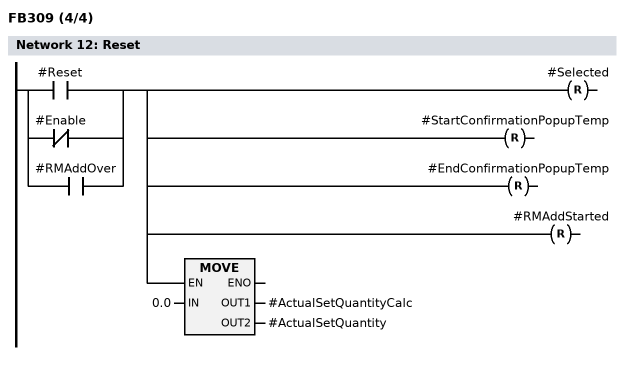
   RUNG wire#powerrail
      Contact( #Reset )
      wire#w1
      R_Coil( #Selected )
   END_RUNG
   RUNG wire#powerrail
      I_Contact( #Enable )
   END_RUNG wire#w1
   RUNG wire#powerrail
      Contact( #RMAddOver )
   END_RUNG wire#w1
   RUNG wire#w1
      R_Coil( #StartConfirmationPopupTemp )
   END_RUNG
   RUNG wire#w1
      R_Coil( #EndConfirmationPopupTemp )
   END_RUNG
   RUNG wire#w1
      R_Coil( #RMAddStarted )
   END_RUNG
   RUNG wire#w1
      Move(in := 0.0, out1 => #ActualSetQuantityCalc, out2 => #ActualSetQuantity)
   END_RUNG
   // the same network as SCL:
   IF #Reset OR NOT #Enable OR #RMAddOver THEN
       #Selected := FALSE;
       #StartConfirmationPopupTemp := FALSE;
       #EndConfirmationPopupTemp := FALSE;
       #RMAddStarted := FALSE;
       #ActualSetQuantityCalc := 0.0;
       #ActualSetQuantity := 0.0;
   END_IF;
END_REGION
END_FUNCTION_BLOCK

